ABB RAPID module: Head_Data.mod

MODULE Head_Data
    RECORD breakpoint
        pos Position;
        num Angle;
    ENDRECORD

    RECORD corrorder
        num X_Init;
        num X_StartOffset;
        num X_Depth;
        num X_ReturnLength;
        num Y_StartOffset;
        num Y_Depth;
        num Y_ReturnLength;
        num Z_StartOffset;
        num Z_Depth;
        num Z_ReturnLength;
        num RY_Torch;
        num Y_MoveCorrConnect;
        num Z_MoveCorrConnect;
    ENDRECORD

    RECORD monRobs
        extjoint monExt;
        robjoint monJoint1;
        robjoint monJoint2;
        pose monPose1;
        pose monPose2;
    ENDRECORD

    RECORD edgedata
        pos EdgePos;
        num Height;
        num Breadth;
        num HoleSize;
        num Thickness;
        num AngleHeight;
        num AngleWidth;
    ENDRECORD

    RECORD jointgroup
        jointtarget Joint1;
        jointtarget Joint2;
        jointtarget JointG;
    ENDRECORD

    RECORD pointgroup
        robtarget Point1;
        robtarget Point2;
        robtarget PointG;
    ENDRECORD

    RECORD targetdata
        robtarget position;
        num cpm;
        num schedule;
        num voltage;
        num wfs;
        num Current;
        num WeaveShape;
        num WeaveType;
        num WeaveLength;
        num WeaveWidth;
        num WeaveDwellLeft;
        num WeaveDwellRight;
        num TrackType;
        num TrackGainY;
        num TrackGainZ;
        num MaxCorr;
        num Bias;
    ENDRECORD

    RECORD torchmotion
        num No;
        num LengthOffset;
        num BreadthOffset;
        num HeightOffset;
        num WorkingAngle;
        num TravelAngle;
        num WeldingSpeed;
        num Schedule;
        num Voltage;
        num FeedingSpeed;
        num Current;
        num WeaveShape;
        num WeaveType;
        num WeaveLength;
        num WeaveWidth;
        num WeaveDwellLeft;
        num WeaveDwellRight;
        num TrackType;
        num TrackGainY;
        num TrackGainZ;
        num MaxCorr;
        num Bias;
    ENDRECORD

    RECORD TcpOrder
        num Tcp_X;
        num Tcp_Y;
        num Tcp_Z;
        num Tcp_Angle;
    ENDRECORD

    PERS corrorder corrStart{10}:=[[25,15,30,10,15,40,10,15,30,15,2,20,20],[50,15,30,10,15,40,10,15,30,15,0,20,20],[25,-15,-30,-10,15,40,10,15,30,15,2,20,20],[0,0,0,0,15,40,10,15,30,15,0,20,20],[0,0,0,0,15,40,10,15,40,15,5,20,20],[25,-15,-30,-10,15,40,10,15,30,15,0,20,20],[999,0,0,0,0,0,0,0,0,0,0,0,0],[999,0,0,0,0,0,0,0,0,0,0,0,0],[999,0,0,0,25,40,10,15,30,30,10,0,0],[999,0,0,0,0,0,0,0,0,0,0,0,0]];
    PERS corrorder corrEnd{10}:=[[25,15,30,10,15,40,10,15,30,15,2,20,20],[50,15,30,10,15,40,10,15,30,15,0,20,20],[25,-15,-30,-10,15,40,10,15,30,15,2,20,20],[0,0,0,0,15,40,10,15,30,15,0,20,20],[0,0,0,0,15,40,10,15,40,15,3,20,20],[25,-15,-30,-10,15,40,10,15,30,15,0,20,20],[999,0,0,0,25,40,10,15,30,10,0,0,0],[999,0,0,0,0,0,0,0,0,0,0,0,0],[0,0,0,0,15,40,10,15,30,15,0,20,20],[0,0,0,0,0,0,0,0,0,0,0,20,20]];

    PERS tooldata tWeld:=[TRUE,[[320.377,0,330.247],[0.92587,0,0.37784,0]],[3.1,[-71.4,3.8,173.2],[1,0,0,0],0.055,0.049,0.005]];
    PERS tooldata tWeld1:=[TRUE,[[319.938,-6.311,330],[0.92587,0.003729,0.377818,-0.009129]],[3.1,[-71.4,3.8,173.2],[1,0,0,0],0.055,0.049,0.005]];
    PERS tooldata tWeld2:=[TRUE,[[319.938,-6.311,330],[0.92587,0.003729,0.377818,-0.009128]],[3.1,[-71.4,3.8,173.2],[1,0,0,0],0.055,0.049,0.005]];

    PERS wobjdata WobjFloor:=[FALSE,TRUE,"",[[-9600,5300,2095],[0,1,0,0]],[[0,0,0],[1,0,0,0]]];
    PERS wobjdata wobjWeldLine:=[FALSE,TRUE,"",[[-9600,5300,2095],[0,1,0,0]],[[19996.2,2781.64,4.14455],[0.708156,0.000193577,0.000194152,-0.706056]]];
    ! [PlanB Moving WObj] ELM_X(갠트리 선형축) 연동 좌표계 — 2026-03-05
    ! 변경 전: ufprog=TRUE(고정), ufmec=""  → 갠트리 이동 시 WObj 미추종
    ! 변경 후: ufprog=FALSE(이동), ufmec="ELM_X" → 갠트리와 함께 WObj 이동
    ! uframe: ELM_X 원점 기준(동일), oframe: 기존 uframe 오프셋을 oframe으로 이전
    PERS wobjdata wobjWeldLine1:=[FALSE,FALSE,"ELM_X",[[0,0,0],[1,0,0,0]],[[488,50,1620],[0,0.707107,-0.707107,0]]];
    PERS wobjdata wobjWeldLine2:=[FALSE,FALSE,"ELM_X",[[0,0,0],[1,0,0,0]],[[488,-50,1620],[0,0.707107,0.707107,0]]];
    PERS wobjdata wobjRotCtr1:=[FALSE,TRUE,"",[[488,0,0],[0,0.707107,-0.707107,0]],[[0,0,0],[1,0,0,0]]];
    PERS wobjdata wobjRotCtr2:=[FALSE,TRUE,"",[[488,0,0],[0,0.707107,0.707107,0]],[[0,0,0],[1,0,0,0]]];

    !!! Mechanical Geometry !!!
    PERS num nLimitX_Negative:=-9600;
    PERS num nLimitX_Positive:=12400;
    PERS num nLimitY_Negative:=0;
    PERS num nLimitY_Positive:=5300;
    PERS num nLimitZ_Negative:=0;
    PERS num nLimitZ_Positive:=2095;
    PERS num nLimitR_Negative:=-90;
    PERS num nLimitR_Positive:=90;

    ! HomeGantry Home Information
    PERS num nHomeGantryX:=-9600;
    PERS num nHomeGantryY:=5300;
    PERS num nHomeGantryZ:=2095;
    PERS num nHomeGantryR:=0;

    PERS num nHomeTcpX:=-9600;
    PERS num nHomeTcpY:=5300;
    PERS num nHomeTcpZ:=2095;

    ! LDS Check Calibration Reference Point
    PERS num nHomeAdjustX:=0;
    PERS num nHomeAdjustY:=0;
    PERS num nHomeAdjustZ:=0;
    PERS num nHomeAdjustR:=0;

    PERS num Camera_Door:=0;
    PERS num Camera_Tilt:=0;

    ! Robot Welding Posture Height
    PERS num nRobHeightMin:=1100;
    PERS num nRobCorrSpaceHeight:=1680;
    PERS num nRobWorkSpaceHeight:=1680;
    PERS num nRobWeldSpaceHeight:=1620;

    PERS num nRotationNegLimit:=-90;
    PERS num nRotationPosLimit:=90;

    !! Variables for Commands
    PERS num nCmdInput:=0;
    PERS num nCmdOutput:=0;
    PERS num nCmdMatch:=0;


    !!! Bool Data !!!
    PERS bool bEnableWeldSkip:=FALSE;
    PERS bool bEnableStartEndPointCorr:=FALSE;
    PERS bool bEnableManualMacro:=FALSE;
    PERS bool bWireTouch1;
    PERS bool bWireTouch2;
    PERS bool bRobSwap:=FALSE;

    !!!!  WarmUp_X !!!!!
    CONST num nWarmUp_Target_X:=10000;

    !commands for move
    CONST num CMD_MOVE_TO_WORLDHOME:=101;
    CONST num CMD_MOVE_TO_MeasurementHOME:=102;
    CONST num CMD_MOVE_TO_TEACHING_All:=104;
    CONST num CMD_MOVE_TO_TEACHING_R1:=105;
    CONST num CMD_MOVE_TO_TEACHING_R2:=106;
    CONST num CMD_MOVE_JOINTS:=107;
    CONST num CMD_MOVE_ABS_GANTRY:=108;
    CONST num CMD_MOVE_INC_GANTRY:=109;
    CONST num CMD_MOVE_TO_ZHOME:=110;
    CONST num CMD_MOVE_TO_nWarmUp:=112;
    CONST num CMD_Tcp_Inspect:=151;

    ! commands for welding
    CONST num CMD_WELD:=200;
    CONST num CMD_WELD_MOTION:=201;
    CONST num CMD_WELD_CORR:=202;
    CONST num CMD_WELD_MOTION_CORR:=203;
    CONST num CMD_WELD_MM:=204;
    CONST num CMD_WELD_MOTION_MM:=205;
    CONST num CMD_WELD_CORR_MM:=206;
    CONST num CMD_WELD_MOTION_CORR_MM:=207;

    !commands for camera actions
    CONST num CMD_CAMERA_DOOR_OPEN:=301;
    CONST num CMD_CAMERA_DOOR_CLOSE:=302;
    CONST num CMD_CAMERA_BLOW_ON:=303;
    CONST num CMD_CAMERA_BLOW_OFF:=304;
    CONST num CMD_CAMERA1_DOOR_OPEN:=311;
    CONST num CMD_CAMERA1_DOOR_CLOSE:=312;
    CONST num CMD_CAMERA2_DOOR_OPEN:=321;
    CONST num CMD_CAMERA2_DOOR_CLOSE:=322;
    CONST num CMD_CAMERA1_BLOW_ON:=313;
    CONST num CMD_CAMERA2_BLOW_ON:=323;
    CONST num CMD_CAMERA1_BLOW_OFF:=314;
    CONST num CMD_CAMERA2_BLOW_OFF:=324;

    !commands for wire processing
    CONST num CMD_WIRE_CUT:=501;
    CONST num CMD_WIRE_CLEAN:=502;
    CONST num CMD_WIRE_BULLSEYE_CHECK:=505;
    CONST num CMD_WIRE_BULLSEYE_UPDATE:=506;
    CONST num CMD_WIRE_ReplacementMode:=507;
    CONST num CMD_ROB1_WIRE_CUT:=511;
    CONST num CMD_ROB2_WIRE_CUT:=512;
    CONST num CMD_WIRE_CLEAN_R1:=513;
    CONST num CMD_WIRE_CLEAN_R2:=514;

    CONST num CMD_GotoTeachingToWirecut:=551;
    CONST num CMD_TeachingToWirecutEntry_R1:=552;
    CONST num CMD_TeachingToWirecut_R1:=553;
    CONST num CMD_ReturnToWirecut:=554;
    CONST num CMD_TeachingToWirecutEntry_R2:=562;
    CONST num CMD_TeachingToWirecut_R2:=563;

    !commands for gantry mechanical origin checking
    CONST num CMD_HOLE_CHECK:=601;
    CONST num CMD_LDS_CHECK:=602;
    CONST num CMD_ManualOrigin_CHECK:=603;

    ! variables related to commands
    PERS num Command:=0;

    !Weld Time
    VAR clock clockWeldTime;
    PERS num nclockWeldTime{2}:=[270.196,134.768];

    !Cycle Time
    VAR clock clockCycleTime;
    PERS num nclockCycleTime:=334.572;

    PERS num nCameraRotationAngle:=0;

    ! variables for welding command
    PERS num nMotionStep:=5;
    PERS num nMotionTotalStep{2}:=[8,8];
    PERS num nMotionStepCount{2}:=[10,10];

    PERS num nLengthWeldLine:=2662.05;
    PERS num nOffsetLength:=0;
    PERS num nOffsetLengthBuffer:=10;

    !! Variables for Welding Macro
    !! sMacro 2nd,3rd Dim: (1: Open, 2: Snip, 3: Welding, 4: Continued, 5: Divied, 8:MergeStart, 9:MergeEnd)
    PERS string stMacro{2}:=["244","244"];
    PERS string stMacroBuffer_{2};
    PERS num nMacro100{2}:=[2,2];
    PERS num nMacro010{2}:=[4,4];
    PERS num nMacro001{2}:=[4,4];
    PERS num nMacro{2}:=[244,244];

    PERS num nMotionStartStepLast{2}:=[4,4];
    PERS num nMotionEndStepLast{2}:=[4,4];
    PERS num nRunningStep{2}:=[40,40];

    PERS edgedata edgeStart{2}:=[[[20002.2,2781.66,4.15085],50,50,0,12,0,0],[[19990.2,2781.62,4.13825],50,50,0,12,0,0]];
    PERS edgedata edgeEnd{2}:=[[[20010.1,119.623,2.69116],50,50,0,12,0,0],[[19998.1,119.588,2.67856],50,50,0,12,0,0]];

    PERS pos posNull:=[0,0,0];
    PERS pos posStart:=[19996.4,2781.64,5.3429];
    PERS pos posStartLast:=[19996.4,2781.64,5.3429];
    PERS num nStartThick:=14.0106;
    PERS pos posEnd:=[20000.3,119.594,0.735352];
    PERS pos posEndLast:=[20000.3,119.594,0.735352];
    PERS num nEndThick:=13.2815;

    PERS breakpoint BreakPoints{10}:=[[[0,0,0],0],[[0,0,0],0],[[0,0,0],0],[[0,0,0],0],[[0,0,0],0],[[0,0,0],0],[[0,0,0],0],[[0,0,0],0],[[0,0,0],0],[[0,0,0],0]];

    ! data for z pos optimization [move,enter,exit]
    PERS num nMaxPartHeightNearArray{3}:=[300,300,300];

    PERS num nTempAdjustGantryZ;

    !!! Variable for correction weldline start & end Pos !!!
    CONST bool bStart:=TRUE;
    CONST bool bEnd:=FALSE;
    PERS bool bCorrectionOk:=FALSE;
    PERS bool bPlateTiltedRx:=FALSE;
    PERS robtarget pSearchStart:=[[-15,6.31316,14.5561],[0.208209,0.745508,-0.572049,0.271343],[0,0,0,1],[9E+09,9E+09,9E+09,9E+09,9E+09,9E+09]];
    PERS robtarget pSearchEnd:=[[15,6.31316,14.5561],[0.208209,0.745508,-0.572049,0.271343],[0,0,0,1],[9E+09,9E+09,9E+09,9E+09,9E+09,9E+09]];
    PERS num nCorrZ_Store:=5.43813;
    PERS num nCorrY_Store:=1.20374;
    PERS num nCorrX_Store:=-5.98633;
    PERS num nCorrFailOffs:=0;
    PERS pos pCorredPosBuffer:=[13.5035,6.32969,14.5309];
    PERS pos pCorredStartPos{2}:=[[2086.6,5904.59,39.6865],[2086.6,5904.59,39.6865]];
    PERS pos pCorredEndPos{2}:=[[2082.19,4521.61,35.0346],[2086.6,5904.59,39.6865]];
    PERS pos pCorredSplitPos:=[2082.19,4521.61,35.0346];

    PERS bool bWeldLineLengthCalc:=FALSE;
    PERS bool bMoveGantry:=FALSE;

    !! Variables for Position of Gantry Move
    PERS extjoint extGantryPos:=[13750,2300,2100,0,0,13750];

    !!! RoboTarget !!!
    CONST robtarget pNull:=[[0,0,0],[1,0,0,0],[0,0,0,0],[9E+09,9E+09,9E+09,9E+09,9E+09,9E+09]];
    CONST robtarget pHome:=[[423.10464973,-0.304,-470.07267919],[0.342020143,0,-0.939692621,0],[0,0,-1,0],[0,0,0,9E+09,9E+09,9E+09]];

    PERS robtarget pReadyConf{2}:=[[[200.384,-150.531,462.112],[0.16437,-0.687406,-0.687732,-0.165769],[0,-1,0,1],[-8705.17,-8705.17,300.411,482.178,9E+09,9E+09]],[[200.384,-150.531,462.112],[0.16437,-0.687406,-0.687732,-0.165769],[0,-1,0,1],[-8705.17,-8705.17,300.411,482.178,9E+09,9E+09]]];
    PERS robtarget pTargetWeldArray{30}:=[[[-5,5,5],[0.307623,-0.549545,-0.742667,-0.227629],[0,0,0,0],[1400,1400,1200,0,9E+9,9E+9]],[[-5,-6,5],[0.307623,-0.549545,-0.742667,-0.227629],[0,0,0,0],[1400,1400,1200,0,9E+9,9E+9]],[[4,-3,5],[0.307623,-0.549545,-0.742667,-0.227629],[0,0,0,0],[1400,1400,1200,0,9E+9,9E+9]],[[200,-3,5],[0.270598,-0.653282,-0.653282,-0.270598],[0,0,0,0],[1400,1400,1200,0,9E+9,9E+9]],[[800,-3,5],[0.270598,-0.653282,-0.653282,-0.270598],[0,0,0,0],[1400,1400,1800,0,9E+9,9E+9]],[[951,-3,5],[0.270598,-0.653282,-0.653282,-0.270598],[0,0,0,0],[1400,1400,1800,0,9E+9,9E+9]],[[986,-3,5],[0.270598,-0.653282,-0.653282,-0.270598],[0,0,0,0],[1400,1400,1800,0,9E+9,9E+9]],[[1002,-3,5],[0.227629,-0.742667,-0.549545,-0.307623],[0,0,0,0],[1400,1400,1800,0,9E+9,9E+9]],[[1005,-6,5],[0.227629,-0.742667,-0.549545,-0.307623],[0,0,0,0],[1400,1400,1800,0,9E+9,9E+9]],[[1005,7,5],[0.227629,-0.742667,-0.549545,-0.307623],[0,0,0,0],[1400,1400,1800,0,9E+9,9E+9]],
                                         [[1005,-6,5],[0.227629,-0.742667,-0.549545,-0.307623],[0,0,0,0],[1400,1400,1800,0,9E+9,9E+9]],[[951,-3,5],[0.270598,-0.653282,-0.653282,-0.270598],[0,0,0,0],[1400,1400,1800,0,9E+9,9E+9]],[[0,0,0],[1,0,0,0],[0,0,0,0],[0,0,0,0,9E+9,9E+9]],[[0,0,0],[1,0,0,0],[0,0,0,0],[0,0,0,0,9E+9,9E+9]],[[0,0,0],[1,0,0,0],[0,0,0,0],[0,0,0,0,9E+9,9E+9]],[[0,0,0],[1,0,0,0],[0,0,0,0],[0,0,0,0,9E+9,9E+9]],[[0,0,0],[1,0,0,0],[0,0,0,0],[0,0,0,0,9E+9,9E+9]],[[0,0,0],[1,0,0,0],[0,0,0,0],[0,0,0,0,9E+9,9E+9]],[[0,0,0],[1,0,0,0],[0,0,0,0],[0,0,0,0,9E+9,9E+9]],[[0,0,0],[1,0,0,0],[0,0,0,0],[0,0,0,0,9E+9,9E+9]],
                                         [[0,0,0],[1,0,0,0],[0,0,0,0],[0,0,0,0,9E+9,9E+9]],[[0,0,0],[1,0,0,0],[0,0,0,0],[0,0,0,0,9E+9,9E+9]],[[0,0,0],[1,0,0,0],[0,0,0,0],[0,0,0,0,9E+9,9E+9]],[[0,0,0],[1,0,0,0],[0,0,0,0],[0,0,0,0,9E+9,9E+9]],[[0,0,0],[1,0,0,0],[0,0,0,0],[0,0,0,0,9E+9,9E+9]],[[0,0,0],[1,0,0,0],[0,0,0,0],[0,0,0,0,9E+9,9E+9]],[[0,0,0],[1,0,0,0],[0,0,0,0],[0,0,0,0,9E+9,9E+9]],[[0,0,0],[1,0,0,0],[0,0,0,0],[0,0,0,0,9E+9,9E+9]],[[0,0,0],[1,0,0,0],[0,0,0,0],[0,0,0,0,9E+9,9E+9]],[[0,0,0],[1,0,0,0],[0,0,0,0],[0,0,0,0,9E+9,9E+9]]];

    !!! Joint Target !!!
    PERS jointtarget jNull:=[[0,0,0,0,0,0],[0,0,0,0,9E+09,0]];
    PERS jointtarget jHomeJoint:=[[9E+09,9E+09,9E+09,9E+09,9E+09,9E+09],[8000,5300,0,0,9E+09,8000]];
    PERS jointgroup jgHomeJoint:=[[[90,90,-45,0,20,0],[9E+09,9E+09,9E+09,9E+09,9E+09,9E+09]],[[90,90,-45,0,20,0],[9E+09,9E+09,9E+09,9E+09,9E+09,9E+09]],[[9E+09,9E+09,9E+09,9E+09,9E+09,9E+09],[8000,5300,0,0,9E+09,8000]]];
    PERS jointtarget jHomeJointBackup:=[[9E+09,9E+09,9E+09,9E+09,9E+09,9E+09],[0,0,6000,500,9E+09,9E+09]];
    PERS jointtarget jRepairJoint:=[[9E+09,9E+09,9E+09,9E+09,9E+09,9E+09],[0,0,6000,500,9E+09,9E+09]];
    PERS jointtarget jMoveReady:=[[9E+9,9E+9,9E+9,9E+9,9E+9,9E+9],[-8707.81,-8707.8,1477.15,0,9E+9,9E+9]];

    PERS jointtarget jJointStepArray{10}:=[[[0,0,0,0,0,0],[0,0,0,0,0,0]],[[0,0,0,0,0,0],[0,0,0,0,0,0]],[[0,0,0,0,0,0],[0,0,0,0,0,0]],[[0,0,0,0,0,0],[0,0,0,0,0,0]],[[0,0,0,0,0,0],[0,0,0,0,0,0]],[[0,-95,65,0,-35,0],[0,0,0,0,0,0]],[[0,0,0,0,0,0],[0,0,0,0,0,0]],[[0,0,0,0,0,0],[0,0,0,0,0,0]],[[0,0,0,0,0,0],[0,0,0,0,0,0]],[[0,-46.86,14,0,-57.52,1.03],[0,0,0,0,0,0]]];

    PERS jointtarget jWeldPos{40}:=[[[0,0,0,0,0,0],[0,0,0,0,9E+09,9E+09]],[[0,0,0,0,0,0],[0,0,0,0,9E+09,9E+09]],[[0,0,0,0,0,0],[0,0,0,0,9E+09,9E+09]],[[0,0,0,0,0,0],[0,0,0,0,9E+09,9E+09]],[[0,0,0,0,0,0],[0,0,0,0,9E+09,9E+09]],[[0,0,0,0,0,0],[0,0,0,0,9E+09,9E+09]],[[0,0,0,0,0,0],[0,0,0,0,9E+09,9E+09]],[[0,0,0,0,0,0],[0,0,0,0,9E+09,9E+09]],[[0,0,0,0,0,0],[0,0,0,0,9E+09,9E+09]],[[0,0,0,0,0,0],[0,0,0,0,9E+09,9E+09]],[[0,0,0,0,0,0],[0,0,0,0,9E+09,9E+09]],[[0,0,0,0,0,0],[0,0,0,0,9E+09,9E+09]],[[0,0,0,0,0,0],[0,0,0,0,9E+09,9E+09]],[[0,0,0,0,0,0],[0,0,0,0,9E+09,9E+09]],[[0,0,0,0,0,0],[0,0,0,0,9E+09,9E+09]],[[0,0,0,0,0,0],[0,0,0,0,9E+09,9E+09]],[[0,0,0,0,0,0],[0,0,0,0,9E+09,9E+09]],[[0,0,0,0,0,0],[0,0,0,0,9E+09,9E+09]],[[0,0,0,0,0,0],[0,0,0,0,9E+09,9E+09]],[[0,0,0,0,0,0],[0,0,0,0,9E+09,9E+09]],[[0,0,0,0,0,0],[0,0,0,0,9E+09,9E+09]],[[0,0,0,0,0,0],[0,0,0,0,9E+09,9E+09]],[[0,0,0,0,0,0],[0,0,0,0,9E+09,9E+09]],[[0,0,0,0,0,0],[0,0,0,0,9E+09,9E+09]],[[0,0,0,0,0,0],[0,0,0,0,9E+09,9E+09]],[[0,0,0,0,0,0],[0,0,0,0,9E+09,9E+09]],[[0,0,0,0,0,0],[0,0,0,0,9E+09,9E+09]],[[0,0,0,0,0,0],[0,0,0,0,9E+09,9E+09]],[[0,0,0,0,0,0],[0,0,0,0,9E+09,9E+09]],[[0,0,0,0,0,0],[0,0,0,0,9E+09,9E+09]],[[0,0,0,0,0,0],[0,0,0,0,9E+09,9E+09]],[[0,0,0,0,0,0],[0,0,0,0,9E+09,9E+09]],[[0,0,0,0,0,0],[0,0,0,0,9E+09,9E+09]],[[0,0,0,0,0,0],[0,0,0,0,9E+09,9E+09]],[[0,0,0,0,0,0],[0,0,0,0,9E+09,9E+09]],[[0,0,0,0,0,0],[0,0,0,0,9E+09,9E+09]],[[0,0,0,0,0,0],[0,0,0,0,9E+09,9E+09]],[[0,0,0,0,0,0],[0,0,0,0,9E+09,9E+09]],[[0,0,0,0,0,0],[0,0,0,0,9E+09,9E+09]],[[0,0,0,0,0,0],[0,0,0,0,9E+09,9E+09]]];
    PERS jointtarget jTest1:=[[9E+09,9E+09,9E+09,9E+09,9E+09,9E+09],[0,0,0,0,9E+09,0]];
    PERS jointtarget jTest2:=[[9E+09,9E+09,9E+09,9E+09,9E+09,9E+09],[0,0,0,0,9E+09,0]];
    PERS jointtarget jTest3:=[[9E+09,9E+09,9E+09,9E+09,9E+09,9E+09],[0,0,0,0,9E+09,0]];
    PERS jointtarget jTest4:=[[9E+09,9E+09,9E+09,9E+09,9E+09,9E+09],[0,0,0,0,9E+09,0]];

    !!! Variables for macroReference !!!
    PERS torchmotion macroAutoStartA{2,10}:=[[[1,0,-2,2,50,0,60,5,36.8,230,380,1,2,2,1.5,1,1,0,0,0,0,0],[2,1,-2,2,50,0,60,5,36.8,230,380,1,2,2,1.5,1,1,0,0,0,0,0],[3,2,-2,2,50,0,60,5,36.8,230,380,1,2,2,1.5,1,1,0,0,0,0,0],[4,3,-2,2,50,0,60,5,36.8,230,380,1,2,2,1.5,1,1,0,0,0,0,0],[999,1,1,1,1,1,1,1,1,1,1,1,1,1,1,1,1,1,1,1,1,1],[1,1,1,1,1,1,1,1,1,1,1,1,1,1,1,1,1,1,1,1,1,1],[1,1,1,1,1,1,1,1,1,1,1,1,1,1,1,1,1,1,1,1,1,1],[1,1,1,1,1,1,1,1,1,1,1,1,1,1,1,1,1,1,1,1,1,1],[1,1,1,1,1,1,1,1,1,1,1,1,1,1,1,1,1,1,1,1,1,1],[1,1,1,1,1,1,1,1,1,1,1,1,1,1,1,1,1,1,1,1,1,1]],[[1,0,-3,2,50,0,60,5,36.3,232,360,1,2,2,1.5,1,1,0,0,0,0,0],[2,1,-3,2,50,0,60,5,36.3,232,360,1,2,2,1.5,1,1,0,0,0,0,0],[3,2,-3,2,50,0,60,5,36.3,232,360,1,2,2,1.5,1,1,0,0,0,0,0],[4,3,-3,2,50,0,60,5,36.3,232,360,1,2,2,1.5,1,1,0,0,0,0,0],[999,1,1,1,1,1,1,1,1,1,1,1,1,1,1,1,1,1,1,1,1,1],[1,1,1,1,1,1,1,1,1,1,1,1,1,1,1,1,1,1,1,1,1,1],[1,1,1,1,1,1,1,1,1,1,1,1,1,1,1,1,1,1,1,1,1,1],[1,1,1,1,1,1,1,1,1,1,1,1,1,1,1,1,1,1,1,1,1,1],[1,1,1,1,1,1,1,1,1,1,1,1,1,1,1,1,1,1,1,1,1,1],[1,1,1,1,1,1,1,1,1,1,1,1,1,1,1,1,1,1,1,1,1,1]]];
    PERS torchmotion macroAutoStartB{2,10}:=[[[1,0,-2,2,50,0,60,5,36.8,230,380,1,2,2,1.5,1,1,0,0,0,0,0],[2,1,-2,2,50,0,60,5,36.8,230,380,1,2,2,1.5,1,1,0,0,0,0,0],[3,2,-2,2,50,0,60,5,36.8,230,380,1,2,2,1.5,1,1,0,0,0,0,0],[4,3,-2,2,50,0,60,5,36.8,230,380,1,2,2,1.5,1,1,0,0,0,0,0],[999,1,1,1,1,1,1,1,1,1,1,1,1,1,1,1,1,1,1,1,1,1],[1,1,1,1,1,1,1,1,1,1,1,1,1,1,1,1,1,1,1,1,1,1],[1,1,1,1,1,1,1,1,1,1,1,1,1,1,1,1,1,1,1,1,1,1],[1,1,1,1,1,1,1,1,1,1,1,1,1,1,1,1,1,1,1,1,1,1],[1,1,1,1,1,1,1,1,1,1,1,1,1,1,1,1,1,1,1,1,1,1],[1,1,1,1,1,1,1,1,1,1,1,1,1,1,1,1,1,1,1,1,1,1]],[[1,0,-3,2,50,0,60,5,36.3,232,360,1,2,2,1.5,1,1,0,0,0,0,0],[2,1,-3,2,50,0,60,5,36.3,232,360,1,2,2,1.5,1,1,0,0,0,0,0],[3,2,-3,2,50,0,60,5,36.3,232,360,1,2,2,1.5,1,1,0,0,0,0,0],[4,3,-3,2,50,0,60,5,36.3,232,360,1,2,2,1.5,1,1,0,0,0,0,0],[999,1,1,1,1,1,1,1,1,1,1,1,1,1,1,1,1,1,1,1,1,1],[1,1,1,1,1,1,1,1,1,1,1,1,1,1,1,1,1,1,1,1,1,1],[1,1,1,1,1,1,1,1,1,1,1,1,1,1,1,1,1,1,1,1,1,1],[1,1,1,1,1,1,1,1,1,1,1,1,1,1,1,1,1,1,1,1,1,1],[1,1,1,1,1,1,1,1,1,1,1,1,1,1,1,1,1,1,1,1,1,1],[1,1,1,1,1,1,1,1,1,1,1,1,1,1,1,1,1,1,1,1,1,1]]];
    PERS torchmotion macroAutoEndA{2,10}:=[[[1,-3,-2,2,50,0,60,5,36.8,230,380,1,2,2,1.5,1,1,0,10,20,30,0],[2,-2,-2,2,50,0,60,5,36.8,230,380,1,2,2,1.5,1,1,0,0,0,0,0],[3,-1,-2,2,50,0,60,5,36.8,230,380,1,2,2,1.5,1,1,0,0,0,0,0],[4,0,-2,2,50,0,60,5,36.8,230,380,1,2,2,1.5,1,1,0,0,0,0,0],[999,1,1,1,1,1,1,1,1,1,1,1,1,1,1,1,1,1,1,1,1,1],[1,1,1,1,1,1,1,1,1,1,1,1,1,1,1,1,1,1,1,1,1,1],[1,1,1,1,1,1,1,1,1,1,1,1,1,1,1,1,1,1,1,1,1,1],[1,1,1,1,1,1,1,1,1,1,1,1,1,1,1,1,1,1,1,1,1,1],[1,1,1,1,1,1,1,1,1,1,1,1,1,1,1,1,1,1,1,1,1,1],[1,1,1,1,1,1,1,1,1,1,1,1,1,1,1,1,1,1,1,1,1,1]],[[1,-3,-3,2,50,0,60,5,36.3,232,360,1,2,2,1.5,1,1,0,10,20,30,0],[2,-2,-3,2,50,0,60,5,36.3,232,360,1,2,2,1.5,1,1,0,0,0,0,0],[3,-1,-2,2,50,0,60,5,36.3,232,360,1,2,2,1.5,1,1,0,0,0,0,0],[4,0,-2,2,50,0,60,5,36.3,232,360,1,2,2,1.5,1,1,0,0,0,0,0],[999,1,1,1,1,1,1,1,1,1,1,1,1,1,1,1,1,1,1,1,1,1],[1,1,1,1,1,1,1,1,1,1,1,1,1,1,1,1,1,1,1,1,1,1],[1,1,1,1,1,1,1,1,1,1,1,1,1,1,1,1,1,1,1,1,1,1],[1,1,1,1,1,1,1,1,1,1,1,1,1,1,1,1,1,1,1,1,1,1],[1,1,1,1,1,1,1,1,1,1,1,1,1,1,1,1,1,1,1,1,1,1],[1,1,1,1,1,1,1,1,1,1,1,1,1,1,1,1,1,1,1,1,1,1]]];
    PERS torchmotion macroAutoEndB{2,10}:=[[[1,-3,-2,2,50,0,60,5,36.8,230,380,1,2,2,1.5,1,1,0,10,20,30,0],[2,-2,-2,2,50,0,60,5,36.8,230,380,1,2,2,1.5,1,1,0,0,0,0,0],[3,-1,-2,2,50,0,60,5,36.8,230,380,1,2,2,1.5,1,1,0,0,0,0,0],[4,0,-2,2,50,0,60,5,36.8,230,380,1,2,2,1.5,1,1,0,0,0,0,0],[999,1,1,1,1,1,1,1,1,1,1,1,1,1,1,1,1,1,1,1,1,1],[1,1,1,1,1,1,1,1,1,1,1,1,1,1,1,1,1,1,1,1,1,1],[1,1,1,1,1,1,1,1,1,1,1,1,1,1,1,1,1,1,1,1,1,1],[1,1,1,1,1,1,1,1,1,1,1,1,1,1,1,1,1,1,1,1,1,1],[1,1,1,1,1,1,1,1,1,1,1,1,1,1,1,1,1,1,1,1,1,1],[1,1,1,1,1,1,1,1,1,1,1,1,1,1,1,1,1,1,1,1,1,1]],[[1,-3,-3,2,50,0,60,5,36.3,232,360,1,2,2,1.5,1,1,0,10,20,30,0],[2,-2,-3,2,50,0,60,5,36.3,232,360,1,2,2,1.5,1,1,0,0,0,0,0],[3,-1,-2,2,50,0,60,5,36.3,232,360,1,2,2,1.5,1,1,0,0,0,0,0],[4,0,-2,2,50,0,60,5,36.3,232,360,1,2,2,1.5,1,1,0,0,0,0,0],[999,1,1,1,1,1,1,1,1,1,1,1,1,1,1,1,1,1,1,1,1,1],[1,1,1,1,1,1,1,1,1,1,1,1,1,1,1,1,1,1,1,1,1,1],[1,1,1,1,1,1,1,1,1,1,1,1,1,1,1,1,1,1,1,1,1,1],[1,1,1,1,1,1,1,1,1,1,1,1,1,1,1,1,1,1,1,1,1,1],[1,1,1,1,1,1,1,1,1,1,1,1,1,1,1,1,1,1,1,1,1,1],[1,1,1,1,1,1,1,1,1,1,1,1,1,1,1,1,1,1,1,1,1,1]]];

    PERS torchmotion macroManualStartA{2,10}:=[[[1,0,-2,2,50,0,60,5,36.5,230,380,1,2,2,1.5,1,1,0,0,0,0,0],[2,1,-2,2,50,0,60,5,36.5,230,380,1,2,2,1.5,1,1,0,0,0,0,0],[3,2,-2,2,50,0,60,5,36.5,230,380,1,2,2,1.5,1,1,0,0,0,0,0],[4,3,-2,2,50,0,60,5,36.5,230,380,1,2,2,1.5,1,1,0,0,0,0,0],[999,1,1,1,1,1,1,1,1,1,1,1,1,1,1,1,1,1,1,1,1,1],[1,1,1,1,1,1,1,1,1,1,1,1,1,1,1,1,1,1,1,1,1,1],[1,1,1,1,1,1,1,1,1,1,1,1,1,1,1,1,1,1,1,1,1,1],[1,1,1,1,1,1,1,1,1,1,1,1,1,1,1,1,1,1,1,1,1,1],[1,1,1,1,1,1,1,1,1,1,1,1,1,1,1,1,1,1,1,1,1,1],[1,1,1,1,1,1,1,1,1,1,1,1,1,1,1,1,1,1,1,1,1,1]],[[1,0,-3,2,50,0,60,5,36.3,232,360,1,2,2,1.5,1,1,0,0,0,0,0],[2,1,-3,2,50,0,60,5,36.3,232,360,1,2,2,1.5,1,1,0,0,0,0,0],[3,2,-3,2,50,0,60,5,36.3,232,360,1,2,2,1.5,1,1,0,0,0,0,0],[4,3,-3,2,50,0,60,5,36.3,232,360,1,2,2,1.5,1,1,0,0,0,0,0],[999,1,1,1,1,1,1,1,1,1,1,1,1,1,1,1,1,1,1,1,1,1],[1,1,1,1,1,1,1,1,1,1,1,1,1,1,1,1,1,1,1,1,1,1],[1,1,1,1,1,1,1,1,1,1,1,1,1,1,1,1,1,1,1,1,1,1],[1,1,1,1,1,1,1,1,1,1,1,1,1,1,1,1,1,1,1,1,1,1],[1,1,1,1,1,1,1,1,1,1,1,1,1,1,1,1,1,1,1,1,1,1],[1,1,1,1,1,1,1,1,1,1,1,1,1,1,1,1,1,1,1,1,1,1]]];
    ![[[1,0,-2,2,50,38,60,5,36.5,230,370,1,2,2,2,1,1,0,0,0,0,0],[2,0,-2,2,50,38,60,5,36.5,230,370,1,2,2,2,1,1,0,0,0,0,0],[3,0,-2,2,50,38,60,5,36.5,230,370,1,2,2,2,1,1,0,0,0,0,0],[4,0,-2,2,50,38,60,5,36.5,230,370,1,2,2,2,1,1,0,0,0,0,0],[999,1,1,1,1,1,1,1,1,1,1,1,1,1,1,1,1,1,1,1,1,1],[1,1,1,1,1,1,1,1,1,1,1,1,1,1,1,1,1,1,1,1,1,1],[1,1,1,1,1,1,1,1,1,1,1,1,1,1,1,1,1,1,1,1,1,1],[1,1,1,1,1,1,1,1,1,1,1,1,1,1,1,1,1,1,1,1,1,1],[1,1,1,1,1,1,1,1,1,1,1,1,1,1,1,1,1,1,1,1,1,1],[1,1,1,1,1,1,1,1,1,1,1,1,1,1,1,1,1,1,1,1,1,1]],[[1,0,-2,2,50,38,60,5,36.5,230,360,1,2,2,2,1,1,0,0,0,0,0],[2,0,-2,2,50,38,60,5,36.5,230,360,1,2,2,2,1,1,0,0,0,0,0],[3,0,-2,2,50,38,60,5,36.5,230,360,1,2,2,2,1,1,0,0,0,0,0],[4,0,-2,2,50,38,60,5,36.5,230,360,1,2,2,2,1,1,0,0,0,0,0],[999,1,1,1,1,1,1,1,1,1,1,1,1,1,1,1,1,1,1,1,1,1],[1,1,1,1,1,1,1,1,1,1,1,1,1,1,1,1,1,1,1,1,1,1],[1,1,1,1,1,1,1,1,1,1,1,1,1,1,1,1,1,1,1,1,1,1],[1,1,1,1,1,1,1,1,1,1,1,1,1,1,1,1,1,1,1,1,1,1],[1,1,1,1,1,1,1,1,1,1,1,1,1,1,1,1,1,1,1,1,1,1],[1,1,1,1,1,1,1,1,1,1,1,1,1,1,1,1,1,1,1,1,1,1]]];
    ![[[1,0,-2,2,50,0,60,5,37,230,380,1,2,2,2,1,1,0,0,0,0,0],[2,0,-2,2,50,0,60,5,37,230,380,1,2,2,2,1,1,0,0,0,0,0],[3,0,-2,2,50,0,60,5,37,230,380,1,2,2,2,1,1,0,0,0,0,0],[4,0,-2,2,50,0,60,5,37,230,380,1,2,2,2,1,1,0,0,0,0,0],[999,1,1,1,1,1,1,1,1,1,1,1,1,1,1,1,1,1,1,1,1,1],[1,1,1,1,1,1,1,1,1,1,1,1,1,1,1,1,1,1,1,1,1,1],[1,1,1,1,1,1,1,1,1,1,1,1,1,1,1,1,1,1,1,1,1,1],[1,1,1,1,1,1,1,1,1,1,1,1,1,1,1,1,1,1,1,1,1,1],[1,1,1,1,1,1,1,1,1,1,1,1,1,1,1,1,1,1,1,1,1,1],[1,1,1,1,1,1,1,1,1,1,1,1,1,1,1,1,1,1,1,1,1,1]],[[1,0,-2,2,50,0,60,5,36.5,230,360,1,2,2,2,1,1,0,0,0,0,0],[2,0,-2,2,50,0,60,5,36.5,230,360,1,2,2,2,1,1,0,0,0,0,0],[3,0,-2,2,50,0,60,5,36.5,230,360,1,2,2,2,1,1,0,0,0,0,0],[4,0,-2,2,50,0,60,5,36.5,230,360,1,2,2,2,1,1,0,0,0,0,0],[999,1,1,1,1,1,1,1,1,1,1,1,1,1,1,1,1,1,1,1,1,1],[1,1,1,1,1,1,1,1,1,1,1,1,1,1,1,1,1,1,1,1,1,1],[1,1,1,1,1,1,1,1,1,1,1,1,1,1,1,1,1,1,1,1,1,1],[1,1,1,1,1,1,1,1,1,1,1,1,1,1,1,1,1,1,1,1,1,1],[1,1,1,1,1,1,1,1,1,1,1,1,1,1,1,1,1,1,1,1,1,1],[1,1,1,1,1,1,1,1,1,1,1,1,1,1,1,1,1,1,1,1,1,1]]];
    PERS torchmotion macroManualStartB{2,10}:=[[[1,0,-2,2,50,0,60,5,36.5,230,380,1,2,2,1.5,1,1,0,0,0,0,0],[2,1,-2,2,50,0,60,5,36.5,230,380,1,2,2,1.5,1,1,0,0,0,0,0],[3,2,-2,2,50,0,60,5,36.5,230,380,1,2,2,1.5,1,1,0,0,0,0,0],[4,3,-2,2,50,0,60,5,36.5,230,380,1,2,2,1.5,1,1,0,0,0,0,0],[999,1,1,1,1,1,1,1,1,1,1,1,1,1,1,1,1,1,1,1,1,1],[1,1,1,1,1,1,1,1,1,1,1,1,1,1,1,1,1,1,1,1,1,1],[1,1,1,1,1,1,1,1,1,1,1,1,1,1,1,1,1,1,1,1,1,1],[1,1,1,1,1,1,1,1,1,1,1,1,1,1,1,1,1,1,1,1,1,1],[1,1,1,1,1,1,1,1,1,1,1,1,1,1,1,1,1,1,1,1,1,1],[1,1,1,1,1,1,1,1,1,1,1,1,1,1,1,1,1,1,1,1,1,1]],[[1,0,-3,2,50,0,60,5,36.3,232,360,1,2,2,1.5,1,1,0,0,0,0,0],[2,1,-3,2,50,0,60,5,36.3,232,360,1,2,2,1.5,1,1,0,0,0,0,0],[3,2,-3,2,50,0,60,5,36.3,232,360,1,2,2,1.5,1,1,0,0,0,0,0],[4,3,-3,2,50,0,60,5,36.3,232,360,1,2,2,1.5,1,1,0,0,0,0,0],[999,1,1,1,1,1,1,1,1,1,1,1,1,1,1,1,1,1,1,1,1,1],[1,1,1,1,1,1,1,1,1,1,1,1,1,1,1,1,1,1,1,1,1,1],[1,1,1,1,1,1,1,1,1,1,1,1,1,1,1,1,1,1,1,1,1,1],[1,1,1,1,1,1,1,1,1,1,1,1,1,1,1,1,1,1,1,1,1,1],[1,1,1,1,1,1,1,1,1,1,1,1,1,1,1,1,1,1,1,1,1,1],[1,1,1,1,1,1,1,1,1,1,1,1,1,1,1,1,1,1,1,1,1,1]]];
    ![[[1,0,-2,2,50,0,60,5,37,230,380,1,2,2,2,1,1,0,0,0,0,0],[2,0,-2,2,50,0,60,5,37,230,380,1,2,2,2,1,1,0,0,0,0,0],[3,0,-2,2,50,0,60,5,37,230,380,1,2,2,2,1,1,0,0,0,0,0],[4,0,-2,2,50,0,60,5,37,230,380,1,2,2,2,1,1,0,0,0,0,0],[999,1,1,1,1,1,1,1,1,1,1,1,1,1,1,1,1,1,1,1,1,1],[1,1,1,1,1,1,1,1,1,1,1,1,1,1,1,1,1,1,1,1,1,1],[1,1,1,1,1,1,1,1,1,1,1,1,1,1,1,1,1,1,1,1,1,1],[1,1,1,1,1,1,1,1,1,1,1,1,1,1,1,1,1,1,1,1,1,1],[1,1,1,1,1,1,1,1,1,1,1,1,1,1,1,1,1,1,1,1,1,1],[1,1,1,1,1,1,1,1,1,1,1,1,1,1,1,1,1,1,1,1,1,1]],[[1,0,-2,2,50,0,60,5,36.5,230,360,1,2,2,2,1,1,0,0,0,0,0],[2,0,-2,2,50,0,60,5,36.5,230,360,1,2,2,2,1,1,0,0,0,0,0],[3,0,-2,2,50,0,60,5,36.5,230,360,1,2,2,2,1,1,0,0,0,0,0],[4,0,-2,2,50,0,60,5,36.5,230,360,1,2,2,2,1,1,0,0,0,0,0],[999,1,1,1,1,1,1,1,1,1,1,1,1,1,1,1,1,1,1,1,1,1],[1,1,1,1,1,1,1,1,1,1,1,1,1,1,1,1,1,1,1,1,1,1],[1,1,1,1,1,1,1,1,1,1,1,1,1,1,1,1,1,1,1,1,1,1],[1,1,1,1,1,1,1,1,1,1,1,1,1,1,1,1,1,1,1,1,1,1],[1,1,1,1,1,1,1,1,1,1,1,1,1,1,1,1,1,1,1,1,1,1],[1,1,1,1,1,1,1,1,1,1,1,1,1,1,1,1,1,1,1,1,1,1]]];
    ![[[1,0,-2,2,50,38,60,5,36.5,230,370,1,2,2,2,1,1,0,0,0,0,0],[2,0,-2,2,50,38,60,5,36.5,230,370,1,2,2,2,1,1,0,0,0,0,0],[3,0,-2,2,50,38,60,5,36.5,230,370,1,2,2,2,1,1,0,0,0,0,0],[4,0,-2,2,50,38,60,5,36.5,230,370,1,2,2,2,1,1,0,0,0,0,0],[999,1,1,1,1,1,1,1,1,1,1,1,1,1,1,1,1,1,1,1,1,1],[1,1,1,1,1,1,1,1,1,1,1,1,1,1,1,1,1,1,1,1,1,1],[1,1,1,1,1,1,1,1,1,1,1,1,1,1,1,1,1,1,1,1,1,1],[1,1,1,1,1,1,1,1,1,1,1,1,1,1,1,1,1,1,1,1,1,1],[1,1,1,1,1,1,1,1,1,1,1,1,1,1,1,1,1,1,1,1,1,1],[1,1,1,1,1,1,1,1,1,1,1,1,1,1,1,1,1,1,1,1,1,1]],[[1,0,-2,2,50,38,60,5,36.5,230,360,1,2,2,2,1,1,0,0,0,0,0],[2,0,-2,2,50,38,60,5,36.5,230,360,1,2,2,2,1,1,0,0,0,0,0],[3,0,-2,2,50,38,60,5,36.5,230,360,1,2,2,2,1,1,0,0,0,0,0],[4,0,-2,2,50,38,60,5,36.5,230,360,1,2,2,2,1,1,0,0,0,0,0],[999,1,1,1,1,1,1,1,1,1,1,1,1,1,1,1,1,1,1,1,1,1],[1,1,1,1,1,1,1,1,1,1,1,1,1,1,1,1,1,1,1,1,1,1],[1,1,1,1,1,1,1,1,1,1,1,1,1,1,1,1,1,1,1,1,1,1],[1,1,1,1,1,1,1,1,1,1,1,1,1,1,1,1,1,1,1,1,1,1],[1,1,1,1,1,1,1,1,1,1,1,1,1,1,1,1,1,1,1,1,1,1],[1,1,1,1,1,1,1,1,1,1,1,1,1,1,1,1,1,1,1,1,1,1]]];
    PERS torchmotion macroManualEndA{2,10}:=[[[1,-3,-2,2,50,0,60,5,36.5,230,380,1,2,2,1.5,1,1,0,10,20,30,0],[2,-2,-2,2,50,0,60,5,36.5,230,380,1,2,2,1.5,1,1,0,0,0,0,0],[3,-1,-2,2,50,0,60,5,36.5,230,380,1,2,2,1.5,1,1,0,0,0,0,0],[4,0,-2,2,50,0,60,5,36.5,230,380,1,2,2,1.5,1,1,0,0,0,0,0],[999,1,1,1,1,1,1,1,1,1,1,1,1,1,1,1,1,1,1,1,1,1],[1,1,1,1,1,1,1,1,1,1,1,1,1,1,1,1,1,1,1,1,1,1],[1,1,1,1,1,1,1,1,1,1,1,1,1,1,1,1,1,1,1,1,1,1],[1,1,1,1,1,1,1,1,1,1,1,1,1,1,1,1,1,1,1,1,1,1],[1,1,1,1,1,1,1,1,1,1,1,1,1,1,1,1,1,1,1,1,1,1],[1,1,1,1,1,1,1,1,1,1,1,1,1,1,1,1,1,1,1,1,1,1]],[[1,-3,-3,2,50,0,60,5,36.3,232,360,1,2,2,1.5,1,1,0,10,20,30,0],[2,-2,-3,2,50,0,60,5,36.3,232,360,1,2,2,1.5,1,1,0,0,0,0,0],[3,-1,-2,2,50,0,60,5,36.3,232,360,1,2,2,1.5,1,1,0,0,0,0,0],[4,0,-2,2,50,0,60,5,36.3,232,360,1,2,2,1.5,1,1,0,0,0,0,0],[999,1,1,1,1,1,1,1,1,1,1,1,1,1,1,1,1,1,1,1,1,1],[1,1,1,1,1,1,1,1,1,1,1,1,1,1,1,1,1,1,1,1,1,1],[1,1,1,1,1,1,1,1,1,1,1,1,1,1,1,1,1,1,1,1,1,1],[1,1,1,1,1,1,1,1,1,1,1,1,1,1,1,1,1,1,1,1,1,1],[1,1,1,1,1,1,1,1,1,1,1,1,1,1,1,1,1,1,1,1,1,1],[1,1,1,1,1,1,1,1,1,1,1,1,1,1,1,1,1,1,1,1,1,1]]];
    ![[[1,0,-2,2,50,-38,60,5,36.5,230,370,1,2,2,2,1,1,0,0,0,0,0],[2,0,-2,2,50,-38,60,5,36.5,230,370,1,2,2,2,1,1,0,0,0,0,0],[3,0,-2,2,50,-38,60,5,36.5,230,370,1,2,2,2,1,1,0,0,0,0,0],[4,0,-2,2,50,-38,60,5,36.5,230,370,1,2,2,2,1,1,0,0,0,0,0],[999,1,1,1,1,1,1,1,1,1,1,1,1,1,1,1,1,1,1,1,1,1],[1,1,1,1,1,1,1,1,1,1,1,1,1,1,1,1,1,1,1,1,1,1],[1,1,1,1,1,1,1,1,1,1,1,1,1,1,1,1,1,1,1,1,1,1],[1,1,1,1,1,1,1,1,1,1,1,1,1,1,1,1,1,1,1,1,1,1],[1,1,1,1,1,1,1,1,1,1,1,1,1,1,1,1,1,1,1,1,1,1],[1,1,1,1,1,1,1,1,1,1,1,1,1,1,1,1,1,1,1,1,1,1]],[[1,0,-2,2,50,-38,60,5,36.5,230,360,1,2,2,2,1,1,0,0,0,0,0],[2,0,-2,2,50,-38,60,5,36.5,230,360,1,2,2,2,1,1,0,0,0,0,0],[3,0,-2,2,50,-38,60,5,36.5,230,360,1,2,2,2,1,1,0,0,0,0,0],[4,0,-2,2,50,-38,60,5,36.5,230,360,1,2,2,2,1,1,0,0,0,0,0],[999,1,1,1,1,1,1,1,1,1,1,1,1,1,1,1,1,1,1,1,1,1],[1,1,1,1,1,1,1,1,1,1,1,1,1,1,1,1,1,1,1,1,1,1],[1,1,1,1,1,1,1,1,1,1,1,1,1,1,1,1,1,1,1,1,1,1],[1,1,1,1,1,1,1,1,1,1,1,1,1,1,1,1,1,1,1,1,1,1],[1,1,1,1,1,1,1,1,1,1,1,1,1,1,1,1,1,1,1,1,1,1],[1,1,1,1,1,1,1,1,1,1,1,1,1,1,1,1,1,1,1,1,1,1]]];
    ![[[1,0,-2,2,50,0,60,5,37,230,380,1,2,2,2,1,1,0,0,0,0,0],[2,0,-2,2,50,0,60,5,37,230,380,1,2,2,2,1,1,0,0,0,0,0],[3,0,-2,2,50,0,60,5,37,230,380,1,2,2,2,1,1,0,0,0,0,0],[4,0,-2,2,50,0,60,5,37,230,380,1,2,2,2,1,1,0,0,0,0,0],[999,1,1,1,1,1,1,1,1,1,1,1,1,1,1,1,1,1,1,1,1,1],[1,1,1,1,1,1,1,1,1,1,1,1,1,1,1,1,1,1,1,1,1,1],[1,1,1,1,1,1,1,1,1,1,1,1,1,1,1,1,1,1,1,1,1,1],[1,1,1,1,1,1,1,1,1,1,1,1,1,1,1,1,1,1,1,1,1,1],[1,1,1,1,1,1,1,1,1,1,1,1,1,1,1,1,1,1,1,1,1,1],[1,1,1,1,1,1,1,1,1,1,1,1,1,1,1,1,1,1,1,1,1,1]],[[1,0,-2,2,50,0,60,5,36.5,230,360,1,2,2,2,1,1,0,0,0,0,0],[2,0,-2,2,50,0,60,5,36.5,230,360,1,2,2,2,1,1,0,0,0,0,0],[3,0,-2,2,50,0,60,5,36.5,230,360,1,2,2,2,1,1,0,0,0,0,0],[4,0,-2,2,50,0,60,5,36.5,230,360,1,2,2,2,1,1,0,0,0,0,0],[999,1,1,1,1,1,1,1,1,1,1,1,1,1,1,1,1,1,1,1,1,1],[1,1,1,1,1,1,1,1,1,1,1,1,1,1,1,1,1,1,1,1,1,1],[1,1,1,1,1,1,1,1,1,1,1,1,1,1,1,1,1,1,1,1,1,1],[1,1,1,1,1,1,1,1,1,1,1,1,1,1,1,1,1,1,1,1,1,1],[1,1,1,1,1,1,1,1,1,1,1,1,1,1,1,1,1,1,1,1,1,1],[1,1,1,1,1,1,1,1,1,1,1,1,1,1,1,1,1,1,1,1,1,1]]];
    PERS torchmotion macroManualEndB{2,10}:=[[[1,-3,-2,2,50,0,60,5,36.5,230,380,1,2,2,1.5,1,1,0,10,20,30,0],[2,-2,-2,2,50,0,60,5,36.5,230,380,1,2,2,1.5,1,1,0,0,0,0,0],[3,-1,-2,2,50,0,60,5,36.5,230,380,1,2,2,1.5,1,1,0,0,0,0,0],[4,0,-2,2,50,0,60,5,36.5,230,380,1,2,2,1.5,1,1,0,0,0,0,0],[999,1,1,1,1,1,1,1,1,1,1,1,1,1,1,1,1,1,1,1,1,1],[1,1,1,1,1,1,1,1,1,1,1,1,1,1,1,1,1,1,1,1,1,1],[1,1,1,1,1,1,1,1,1,1,1,1,1,1,1,1,1,1,1,1,1,1],[1,1,1,1,1,1,1,1,1,1,1,1,1,1,1,1,1,1,1,1,1,1],[1,1,1,1,1,1,1,1,1,1,1,1,1,1,1,1,1,1,1,1,1,1],[1,1,1,1,1,1,1,1,1,1,1,1,1,1,1,1,1,1,1,1,1,1]],[[1,-3,-3,2,50,0,60,5,36.3,232,360,1,2,2,1.5,1,1,0,10,20,30,0],[2,-2,-3,2,50,0,60,5,36.3,232,360,1,2,2,1.5,1,1,0,0,0,0,0],[3,-1,-2,2,50,0,60,5,36.3,232,360,1,2,2,1.5,1,1,0,0,0,0,0],[4,0,-2,2,50,0,60,5,36.3,232,360,1,2,2,1.5,1,1,0,0,0,0,0],[999,1,1,1,1,1,1,1,1,1,1,1,1,1,1,1,1,1,1,1,1,1],[1,1,1,1,1,1,1,1,1,1,1,1,1,1,1,1,1,1,1,1,1,1],[1,1,1,1,1,1,1,1,1,1,1,1,1,1,1,1,1,1,1,1,1,1],[1,1,1,1,1,1,1,1,1,1,1,1,1,1,1,1,1,1,1,1,1,1],[1,1,1,1,1,1,1,1,1,1,1,1,1,1,1,1,1,1,1,1,1,1],[1,1,1,1,1,1,1,1,1,1,1,1,1,1,1,1,1,1,1,1,1,1]]];
    ![[[1,0,-2,2,50,0,60,5,37,230,380,1,2,2,2,1,1,0,0,0,0,0],[2,0,-2,2,50,0,60,5,37,230,380,1,2,2,2,1,1,0,0,0,0,0],[3,0,-2,2,50,0,60,5,37,230,380,1,2,2,2,1,1,0,0,0,0,0],[4,0,-2,2,50,0,60,5,37,230,380,1,2,2,2,1,1,0,0,0,0,0],[999,1,1,1,1,1,1,1,1,1,1,1,1,1,1,1,1,1,1,1,1,1],[1,1,1,1,1,1,1,1,1,1,1,1,1,1,1,1,1,1,1,1,1,1],[1,1,1,1,1,1,1,1,1,1,1,1,1,1,1,1,1,1,1,1,1,1],[1,1,1,1,1,1,1,1,1,1,1,1,1,1,1,1,1,1,1,1,1,1],[1,1,1,1,1,1,1,1,1,1,1,1,1,1,1,1,1,1,1,1,1,1],[1,1,1,1,1,1,1,1,1,1,1,1,1,1,1,1,1,1,1,1,1,1]],[[1,0,-2,2,50,0,60,5,36.5,230,360,1,2,2,2,1,1,0,0,0,0,0],[2,0,-2,2,50,0,60,5,36.5,230,360,1,2,2,2,1,1,0,0,0,0,0],[3,0,-2,2,50,0,60,5,36.5,230,360,1,2,2,2,1,1,0,0,0,0,0],[4,0,-2,2,50,0,60,5,36.5,230,360,1,2,2,2,1,1,0,0,0,0,0],[999,1,1,1,1,1,1,1,1,1,1,1,1,1,1,1,1,1,1,1,1,1],[1,1,1,1,1,1,1,1,1,1,1,1,1,1,1,1,1,1,1,1,1,1],[1,1,1,1,1,1,1,1,1,1,1,1,1,1,1,1,1,1,1,1,1,1],[1,1,1,1,1,1,1,1,1,1,1,1,1,1,1,1,1,1,1,1,1,1],[1,1,1,1,1,1,1,1,1,1,1,1,1,1,1,1,1,1,1,1,1,1],[1,1,1,1,1,1,1,1,1,1,1,1,1,1,1,1,1,1,1,1,1,1]]];
    ![[[1,0,-2,2,50,-38,60,5,36.5,230,370,1,2,2,2,1,1,0,0,0,0,0],[2,0,-2,2,50,-38,60,5,36.5,230,370,1,2,2,2,1,1,0,0,0,0,0],[3,0,-2,2,50,-38,60,5,36.5,230,370,1,2,2,2,1,1,0,0,0,0,0],[4,0,-2,2,50,-38,60,5,36.5,230,370,1,2,2,2,1,1,0,0,0,0,0],[999,1,1,1,1,1,1,1,1,1,1,1,1,1,1,1,1,1,1,1,1,1],[1,1,1,1,1,1,1,1,1,1,1,1,1,1,1,1,1,1,1,1,1,1],[1,1,1,1,1,1,1,1,1,1,1,1,1,1,1,1,1,1,1,1,1,1],[1,1,1,1,1,1,1,1,1,1,1,1,1,1,1,1,1,1,1,1,1,1],[1,1,1,1,1,1,1,1,1,1,1,1,1,1,1,1,1,1,1,1,1,1],[1,1,1,1,1,1,1,1,1,1,1,1,1,1,1,1,1,1,1,1,1,1]],[[1,0,-2,2,50,-38,60,5,36.5,230,360,1,2,2,2,1,1,0,0,0,0,0],[2,0,-2,2,50,-38,60,5,36.5,230,360,1,2,2,2,1,1,0,0,0,0,0],[3,0,-2,2,50,-38,60,5,36.5,230,360,1,2,2,2,1,1,0,0,0,0,0],[4,0,-2,2,50,-38,60,5,36.5,230,360,1,2,2,2,1,1,0,0,0,0,0],[999,1,1,1,1,1,1,1,1,1,1,1,1,1,1,1,1,1,1,1,1,1],[1,1,1,1,1,1,1,1,1,1,1,1,1,1,1,1,1,1,1,1,1,1],[1,1,1,1,1,1,1,1,1,1,1,1,1,1,1,1,1,1,1,1,1,1],[1,1,1,1,1,1,1,1,1,1,1,1,1,1,1,1,1,1,1,1,1,1],[1,1,1,1,1,1,1,1,1,1,1,1,1,1,1,1,1,1,1,1,1,1],[1,1,1,1,1,1,1,1,1,1,1,1,1,1,1,1,1,1,1,1,1,1]]];

    PERS torchmotion macroStartBuffer1{10}:=[[1,0,-2,2,50,0,60,5,36.8,230,380,1,2,2,1.5,1,1,0,0,0,0,0],[2,1,-2,2,50,0,60,5,36.8,230,380,1,2,2,1.5,1,1,0,0,0,0,0],[3,2,-2,2,50,0,60,5,36.8,230,380,1,2,2,1.5,1,1,0,0,0,0,0],[4,3,-2,2,50,0,60,5,36.8,230,380,1,2,2,1.5,1,1,0,0,0,0,0],[999,1,1,1,1,1,1,1,1,1,1,1,1,1,1,1,1,1,1,1,1,1],[1,1,1,1,1,1,1,1,1,1,1,1,1,1,1,1,1,1,1,1,1,1],[1,1,1,1,1,1,1,1,1,1,1,1,1,1,1,1,1,1,1,1,1,1],[1,1,1,1,1,1,1,1,1,1,1,1,1,1,1,1,1,1,1,1,1,1],[1,1,1,1,1,1,1,1,1,1,1,1,1,1,1,1,1,1,1,1,1,1],[1,1,1,1,1,1,1,1,1,1,1,1,1,1,1,1,1,1,1,1,1,1]];
    PERS torchmotion macroStartBuffer2{10}:=[[1,0,-3,2,50,0,60,5,36.3,232,360,1,2,2,1.5,1,1,0,0,0,0,0],[2,1,-3,2,50,0,60,5,36.3,232,360,1,2,2,1.5,1,1,0,0,0,0,0],[3,2,-3,2,50,0,60,5,36.3,232,360,1,2,2,1.5,1,1,0,0,0,0,0],[4,3,-3,2,50,0,60,5,36.3,232,360,1,2,2,1.5,1,1,0,0,0,0,0],[999,1,1,1,1,1,1,1,1,1,1,1,1,1,1,1,1,1,1,1,1,1],[1,1,1,1,1,1,1,1,1,1,1,1,1,1,1,1,1,1,1,1,1,1],[1,1,1,1,1,1,1,1,1,1,1,1,1,1,1,1,1,1,1,1,1,1],[1,1,1,1,1,1,1,1,1,1,1,1,1,1,1,1,1,1,1,1,1,1],[1,1,1,1,1,1,1,1,1,1,1,1,1,1,1,1,1,1,1,1,1,1],[1,1,1,1,1,1,1,1,1,1,1,1,1,1,1,1,1,1,1,1,1,1]];
    PERS torchmotion macroEndBuffer1{10}:=[[1,-3,-2,2,50,0,60,5,36.8,230,380,1,2,2,1.5,1,1,0,10,20,30,0],[2,-2,-2,2,50,0,60,5,36.8,230,380,1,2,2,1.5,1,1,0,0,0,0,0],[3,-1,-2,2,50,0,60,5,36.8,230,380,1,2,2,1.5,1,1,0,0,0,0,0],[4,0,-2,2,50,0,60,5,36.8,230,380,1,2,2,1.5,1,1,0,0,0,0,0],[999,1,1,1,1,1,1,1,1,1,1,1,1,1,1,1,1,1,1,1,1,1],[1,1,1,1,1,1,1,1,1,1,1,1,1,1,1,1,1,1,1,1,1,1],[1,1,1,1,1,1,1,1,1,1,1,1,1,1,1,1,1,1,1,1,1,1],[1,1,1,1,1,1,1,1,1,1,1,1,1,1,1,1,1,1,1,1,1,1],[1,1,1,1,1,1,1,1,1,1,1,1,1,1,1,1,1,1,1,1,1,1],[1,1,1,1,1,1,1,1,1,1,1,1,1,1,1,1,1,1,1,1,1,1]];
    PERS torchmotion macroEndBuffer2{10}:=[[1,-3,-3,2,50,0,60,5,36.3,232,360,1,2,2,1.5,1,1,0,10,20,30,0],[2,-2,-3,2,50,0,60,5,36.3,232,360,1,2,2,1.5,1,1,0,0,0,0,0],[3,-1,-2,2,50,0,60,5,36.3,232,360,1,2,2,1.5,1,1,0,0,0,0,0],[4,0,-2,2,50,0,60,5,36.3,232,360,1,2,2,1.5,1,1,0,0,0,0,0],[999,1,1,1,1,1,1,1,1,1,1,1,1,1,1,1,1,1,1,1,1,1],[1,1,1,1,1,1,1,1,1,1,1,1,1,1,1,1,1,1,1,1,1,1],[1,1,1,1,1,1,1,1,1,1,1,1,1,1,1,1,1,1,1,1,1,1],[1,1,1,1,1,1,1,1,1,1,1,1,1,1,1,1,1,1,1,1,1,1],[1,1,1,1,1,1,1,1,1,1,1,1,1,1,1,1,1,1,1,1,1,1],[1,1,1,1,1,1,1,1,1,1,1,1,1,1,1,1,1,1,1,1,1,1]];



    !!! Teaching Pose !!!
    PERS jointtarget jTeachPose10:=[[0,-11.58,-54.61,0,-23.21,0],[9E+09,9E+09,9E+09,9E+09,9E+09,9E+09]];
    PERS jointtarget jTeachPose20:=[[0,-13.77,-51.14,0,-24.5,0],[9E+09,9E+09,9E+09,9E+09,9E+09,9E+09]];
    PERS jointtarget jTeachPose30:=[[0,-5.48,-66.86,0,-35.66,0],[9E+09,9E+09,9E+09,9E+09,9E+09,9E+09]];
    PERS jointtarget jTeachPose40:=[[0,-95,70,0,-35,0],[9E+09,9E+09,9E+09,9E+09,9E+09,9E+09]];

    !!! Wire Cut !!!
    PERS jointtarget jWireCutRdy10:=[[-5.74337,56.5223,-2.36426,0,0,0],[-7805.23,-7805.23,1917.83,1534,9E+09,9E+09]];
    PERS jointtarget jWireCutRdy20:=[[-4.42117,43.9252,29.766,35.9723,-31.0497,-17.7691],[-7805.23,-7805.23,1917.83,1534,9E+09,9E+09]];
    PERS jointtarget jWireCutRdy30:=[[-2.45489,39.2604,46.5236,54.029,-43.8022,-8.52495],[-7805.23,-7805.23,1917.83,1534,9E+09,9E+09]];
    PERS jointtarget jWireCutRdy40:=[[-8.44041,38.4714,56.4802,74.9109,-46.3356,6.60117],[-7805.23,-7805.23,1917.83,1534,9E+09,9E+09]];
    PERS jointtarget jWireCut:=[[-10.3272,38.7931,61.3627,68.3466,-47.9698,13.406],[-7805.23,-7805.23,1917.83,1534,9E+09,9E+09]];
    PERS jointtarget jWireCutRdy50:=[[-8.44041,38.4714,56.4802,74.9108,-46.3356,6.60084],[-7805.23,-7805.23,1917.83,1534,9E+09,9E+09]];
    PERS jointtarget jWireCutRdy60:=[[-4.42128,43.9251,29.766,35.9723,-31.0497,-17.7691],[-7805.23,-7805.23,1917.83,1534,9E+09,9E+09]];
    PERS jointtarget jWireCutRdy70:=[[-5.74337,56.5222,-2.36431,0,0,0],[-7805.23,-7805.23,1917.83,1534,9E+09,9E+09]];

    !!! rNozzle Clean !!!
    PERS jointtarget jNozzleClean10:=[[92.7023,56.7732,-24.6002,-105.292,47.2145,-39.1763],[-7.83472,-7.83523,5212.01,422.601,9E+09,9E+09]];
    PERS jointtarget jNozzleClean20:=[[154.238,56.7746,-24.5971,-105.291,47.2139,-39.1774],[-7.83472,-7.83495,5212.01,422.595,9E+09,9E+09]];
    PERS jointtarget jNozzleClean30:=[[144.266,78.8984,-24.7284,-105.291,47.2139,-39.1774],[-7.83513,-7.83495,5212.01,422.596,9E+09,9E+09]];
    PERS jointtarget jNozzleClean40:=[[136.493,90.5978,-51.7581,-95.8271,39.0251,-59.7871],[-7.83513,-7.83482,5212.01,422.595,9E+09,9E+09]];
    PERS jointtarget jNozzleClean:=[[136.493,90.5979,-51.7581,-95.8269,39.0251,-59.7873],[-7.83513,-7.83495,5212.01,422.595,9E+09,9E+09]];
    PERS jointtarget jNozzleClean50:=[[136.493,90.5979,-51.7581,-95.8269,39.0252,-59.7873],[-7.83513,-7.83495,5212.01,422.595,9E+09,9E+09]];
    PERS jointtarget jNozzleClean60:=[[144.266,78.8983,-24.7285,-105.291,47.2139,-39.1774],[-7.83513,-7.83495,5212.01,422.595,9E+09,9E+09]];
    PERS jointtarget jNozzleClean70:=[[154.238,56.7746,-24.5971,-105.291,47.2139,-39.1774],[-7.83513,-7.83495,5212.01,422.595,9E+09,9E+09]];
    PERS jointtarget jNozzleClean80:=[[92.7023,56.7732,-24.6003,-105.292,47.2145,-39.176],[-7.83472,-7.83523,5212.01,422.601,9E+09,9E+09]];

    PERS jointgroup ManualOrigin_Pos:=[[[90,90,-45,0,20,0],[9E+09,9E+09,9E+09,9E+09,9E+09,9E+09]],[[90,90,-45,0,20,0],[9E+09,9E+09,9E+09,9E+09,9E+09,9E+09]],[[9E+09,9E+09,9E+09,9E+09,9E+09,9E+09],[1391,5300,841,0,9E+09,1391]]];

    PERS robtarget pWeldPosR1{40}:=[[[-3,7,1],[0.307623,-0.549545,-0.742667,-0.227629],[-1,0,0,1],[-8704.03,-8704.03,294.161,1030.31,9E+9,9E+9]],[[-3,7,1],[0.307623,-0.549545,-0.742667,-0.227629],[-1,0,0,1],[-8704.03,-8704.03,294.161,1030.31,9E+9,9E+9]],[[-3,-4.5,1],[0.307623,-0.549545,-0.742667,-0.227629],[-1,0,0,1],[-8704.03,-8704.03,294.161,1030.31,9E+9,9E+9]],[[15,-1,1],[0.307623,-0.549545,-0.742667,-0.227629],[-1,0,0,1],[-8704.03,-8704.03,294.161,1030.34,9E+9,9E+9]],[[200,-1,1],[0.270598,-0.653282,-0.653282,-0.270598],[-1,0,0,1],[-8704.03,-8704.03,294.161,1030.72,9E+9,9E+9]],[[1390,-1.00592,0.996463],[0.270597,-0.653283,-0.653281,-0.270597],[0,0,-1,1],[-8707.81,-8707.8,1477.15,1033.13,9E+9,9E+9]],[[0,0,0],[0,0,0,0],[0,0,0,0],[0,0,0,0,0,0]],[[0,0,0],[0,0,0,0],[0,0,0,0],[0,0,0,0,0,0]],[[0,0,0],[0,0,0,0],[0,0,0,0],[0,0,0,0,0,0]],[[0,0,0],[0,0,0,0],[0,0,0,0],[0,0,0,0,0,0]],[[0,0,0],[0,0,0,0],[0,0,0,0],[0,0,0,0,0,0]],[[0,0,0],[0,0,0,0],[0,0,0,0],[0,0,0,0,0,0]],[[0,0,0],[0,0,0,0],[0,0,0,0],[0,0,0,0,0,0]],[[0,0,0],[0,0,0,0],[0,0,0,0],[0,0,0,0,0,0]],[[0,0,0],[0,0,0,0],[0,0,0,0],[0,0,0,0,0,0]],[[0,0,0],[0,0,0,0],[0,0,0,0],[0,0,0,0,0,0]],[[0,0,0],[0,0,0,0],[0,0,0,0],[0,0,0,0,0,0]],[[0,0,0],[0,0,0,0],[0,0,0,0],[0,0,0,0,0,0]],[[0,0,0],[0,0,0,0],[0,0,0,0],[0,0,0,0,0,0]],[[0,0,0],[0,0,0,0],[0,0,0,0],[0,0,0,0,0,0]],[[0,0,0],[0,0,0,0],[0,0,0,0],[0,0,0,0,0,0]],[[0,0,0],[0,0,0,0],[0,0,0,0],[0,0,0,0,0,0]],[[0,0,0],[0,0,0,0],[0,0,0,0],[0,0,0,0,0,0]],[[0,0,0],[0,0,0,0],[0,0,0,0],[0,0,0,0,0,0]],[[0,0,0],[0,0,0,0],[0,0,0,0],[0,0,0,0,0,0]],[[0,0,0],[0,0,0,0],[0,0,0,0],[0,0,0,0,0,0]],[[0,0,0],[0,0,0,0],[0,0,0,0],[0,0,0,0,0,0]],[[0,0,0],[0,0,0,0],[0,0,0,0],[0,0,0,0,0,0]],[[0,0,0],[0,0,0,0],[0,0,0,0],[0,0,0,0,0,0]],[[0,0,0],[0,0,0,0],[0,0,0,0],[0,0,0,0,0,0]],[[0,0,0],[0,0,0,0],[0,0,0,0],[0,0,0,0,0,0]],[[0,0,0],[0,0,0,0],[0,0,0,0],[0,0,0,0,0,0]],[[0,0,0],[0,0,0,0],[0,0,0,0],[0,0,0,0,0,0]],[[0,0,0],[0,0,0,0],[0,0,0,0],[0,0,0,0,0,0]],[[0,0,0],[0,0,0,0],[0,0,0,0],[0,0,0,0,0,0]],[[0,0,0],[0,0,0,0],[0,0,0,0],[0,0,0,0,0,0]],[[0,0,0],[0,0,0,0],[0,0,0,0],[0,0,0,0,0,0]],[[0,0,0],[0,0,0,0],[0,0,0,0],[0,0,0,0,0,0]],[[0,0,0],[0,0,0,0],[0,0,0,0],[0,0,0,0,0,0]],[[15,-1,1],[0.307623,-0.549545,-0.742667,-0.227629],[-1,0,0,1],[-8704.03,-8704.03,294.161,1030.34,9E+9,9E+9]]];
    PERS robtarget pWeldPosR2{40}:=[[[-3,7,1],[0.307623,-0.549545,-0.742667,-0.227629],[-1,0,0,1],[-8704.03,-8704.03,294.161,1030.31,9E+09,9E+09]],[[-3,7,1],[0.307623,-0.549545,-0.742667,-0.227629],[-1,0,0,1],[-8704.03,-8704.03,294.161,1030.31,9E+09,9E+09]],[[-3,-4.5,1],[0.307623,-0.549545,-0.742667,-0.227629],[-1,0,0,1],[-8704.03,-8704.03,294.161,1030.31,9E+09,9E+09]],[[15,-1,1],[0.307623,-0.549545,-0.742667,-0.227629],[-1,0,0,1],[-8704.03,-8704.03,294.161,1030.34,9E+09,9E+09]],[[200,-1,1],[0.270598,-0.653282,-0.653282,-0.270598],[-1,0,0,1],[-8704.03,-8704.03,294.161,1030.72,9E+09,9E+09]],[[1390,-1.00592,0.996463],[0.270597,-0.653283,-0.653281,-0.270597],[0,0,-1,1],[-8707.81,-8707.8,1477.15,1033.13,9E+09,9E+09]],[[0,0,0],[0,0,0,0],[0,0,0,0],[0,0,0,0,0,0]],[[0,0,0],[0,0,0,0],[0,0,0,0],[0,0,0,0,0,0]],[[0,0,0],[0,0,0,0],[0,0,0,0],[0,0,0,0,0,0]],[[0,0,0],[0,0,0,0],[0,0,0,0],[0,0,0,0,0,0]],[[0,0,0],[0,0,0,0],[0,0,0,0],[0,0,0,0,0,0]],[[0,0,0],[0,0,0,0],[0,0,0,0],[0,0,0,0,0,0]],[[0,0,0],[0,0,0,0],[0,0,0,0],[0,0,0,0,0,0]],[[0,0,0],[0,0,0,0],[0,0,0,0],[0,0,0,0,0,0]],[[0,0,0],[0,0,0,0],[0,0,0,0],[0,0,0,0,0,0]],[[0,0,0],[0,0,0,0],[0,0,0,0],[0,0,0,0,0,0]],[[0,0,0],[0,0,0,0],[0,0,0,0],[0,0,0,0,0,0]],[[0,0,0],[0,0,0,0],[0,0,0,0],[0,0,0,0,0,0]],[[0,0,0],[0,0,0,0],[0,0,0,0],[0,0,0,0,0,0]],[[0,0,0],[0,0,0,0],[0,0,0,0],[0,0,0,0,0,0]],[[0,0,0],[0,0,0,0],[0,0,0,0],[0,0,0,0,0,0]],[[0,0,0],[0,0,0,0],[0,0,0,0],[0,0,0,0,0,0]],[[0,0,0],[0,0,0,0],[0,0,0,0],[0,0,0,0,0,0]],[[0,0,0],[0,0,0,0],[0,0,0,0],[0,0,0,0,0,0]],[[0,0,0],[0,0,0,0],[0,0,0,0],[0,0,0,0,0,0]],[[0,0,0],[0,0,0,0],[0,0,0,0],[0,0,0,0,0,0]],[[0,0,0],[0,0,0,0],[0,0,0,0],[0,0,0,0,0,0]],[[0,0,0],[0,0,0,0],[0,0,0,0],[0,0,0,0,0,0]],[[0,0,0],[0,0,0,0],[0,0,0,0],[0,0,0,0,0,0]],[[0,0,0],[0,0,0,0],[0,0,0,0],[0,0,0,0,0,0]],[[0,0,0],[0,0,0,0],[0,0,0,0],[0,0,0,0,0,0]],[[0,0,0],[0,0,0,0],[0,0,0,0],[0,0,0,0,0,0]],[[0,0,0],[0,0,0,0],[0,0,0,0],[0,0,0,0,0,0]],[[0,0,0],[0,0,0,0],[0,0,0,0],[0,0,0,0,0,0]],[[0,0,0],[0,0,0,0],[0,0,0,0],[0,0,0,0,0,0]],[[0,0,0],[0,0,0,0],[0,0,0,0],[0,0,0,0,0,0]],[[0,0,0],[0,0,0,0],[0,0,0,0],[0,0,0,0,0,0]],[[0,0,0],[0,0,0,0],[0,0,0,0],[0,0,0,0,0,0]],[[0,0,0],[0,0,0,0],[0,0,0,0],[0,0,0,0,0,0]],[[1390,-1,1],[0.270598,-0.653282,-0.653282,-0.270598],[-1,0,0,1],[-8707.8,-8707.8,1477.15,1033.12,9E+09,9E+09]]];
    PERS robtarget pWeldPosG{40};
    PERS speeddata vWeld1{40}:=[[10,200,200,200],[10,200,200,200],[10,200,200,200],[10,200,200,200],[10,200,200,200],[10,200,200,200],[0,0,0,0],[0,0,0,0],[0,0,0,0],[0,0,0,0],[0,0,0,0],[0,0,0,0],[0,0,0,0],[0,0,0,0],[0,0,0,0],[0,0,0,0],[0,0,0,0],[0,0,0,0],[0,0,0,0],[0,0,0,0],[0,0,0,0],[0,0,0,0],[0,0,0,0],[0,0,0,0],[0,0,0,0],[0,0,0,0],[0,0,0,0],[0,0,0,0],[0,0,0,0],[0,0,0,0],[0,0,0,0],[0,0,0,0],[0,0,0,0],[0,0,0,0],[0,0,0,0],[0,0,0,0],[0,0,0,0],[0,0,0,0],[0,0,0,0],[10,200,200,200]];
    PERS speeddata vWeld2{40}:=[[10,200,200,200],[10,200,200,200],[10,200,200,200],[10,200,200,200],[10,200,200,200],[10,200,200,200],[0,0,0,0],[0,0,0,0],[0,0,0,0],[0,0,0,0],[0,0,0,0],[0,0,0,0],[0,0,0,0],[0,0,0,0],[0,0,0,0],[0,0,0,0],[0,0,0,0],[0,0,0,0],[0,0,0,0],[0,0,0,0],[0,0,0,0],[0,0,0,0],[0,0,0,0],[0,0,0,0],[0,0,0,0],[0,0,0,0],[0,0,0,0],[0,0,0,0],[0,0,0,0],[0,0,0,0],[0,0,0,0],[0,0,0,0],[0,0,0,0],[0,0,0,0],[0,0,0,0],[0,0,0,0],[0,0,0,0],[0,0,0,0],[0,0,0,0],[10,200,200,200]];

    !!! Speed Data !!!
    PERS speeddata vTargetSpeed:=[400,300,400,25];
    PERS speeddata vTargetSpeed2:=[9,200,200,25];
    PERS speeddata vWeldEntry:=[100,20,200,25];

    !!! variables for Speed Data !!!
    PERS num nWireCutSpeed:=500;
    PERS num nGantrySpeed:=0;
    PERS num nDryRunSpeed:=2.5;

    !!! Zone Data !!!
    PERS zonedata zTargetZone:=[FALSE,30,5,5,2,1,1];
    PERS zonedata zFineZone:=[TRUE,0,0,0,0,0,0];

    VAR num rotationMaxtrix{3,3};

    ! MoveStepGantryHeight
    PERS num nCurrentGantryHeight:=0;
    PERS num nTargetGantryHeight:=-35.9858;
    PERS num nCalculatedGantryHeight:=0;
    PERS num nGantrySafetyHeight:=-100;
    PERS jointtarget jReadyGantryHeightBuffer:=[[9E+09,9E+09,9E+09,9E+09,9E+09,9E+09],[10404,5130.4,-0.000881434,89.8303,9E+09,10404]];
    PERS num nAngleOfEntry:=0.155838;
    PERS num nAngleRzStore:=-89.8299;
    PERS num nCalculatedHeight:=461.831;

    !!! weld data !!!
    TASK PERS welddata wdArray{40}:=[[10,0,[5,0,36.8,230,0,0,0,0,0],[0,0,0,0,0,0,0,0,0]],[10,0,[5,0,36.8,230,0,0,0,0,0],[0,0,0,0,0,0,0,0,0]],[10,0,[5,0,36.8,230,0,0,0,0,0],[0,0,0,0,0,0,0,0,0]],[10,0,[5,0,36.8,230,0,0,0,0,0],[0,0,0,0,0,0,0,0,0]],[10,0,[5,0,36.8,230,0,0,0,0,0],[0,0,0,0,0,0,0,0,0]],[10,0,[5,0,36.8,230,0,0,0,0,0],[0,0,0,0,0,0,0,0,0]],[10,0,[5,0,36.8,230,0,0,0,0,0],[0,0,0,0,0,0,0,0,0]],[10,0,[5,0,36.8,230,0,0,0,0,0],[0,0,0,0,0,0,0,0,0]],[10,0,[5,0,36.8,230,0,0,0,0,0],[0,0,0,0,0,0,0,0,0]],[10,0,[5,0,36.8,230,0,0,0,0,0],[0,0,0,0,0,0,0,0,0]],[10,0,[5,0,34,210,0,0,0,0,0],[0,0,0,0,0,0,0,0,0]],[10,0,[5,0,34,210,0,0,0,0,0],[0,0,0,0,0,0,0,0,0]],[10,0,[5,0,37.5,270,0,0,0,0,0],[0,0,0,0,0,0,0,0,0]],[10,0,[5,0,37.5,250,0,0,0,0,0],[0,0,0,0,0,0,0,0,0]],[10,0,[5,0,37.5,250,0,0,0,0,0],[0,0,0,0,0,0,0,0,0]],[10,0,[5,0,37.5,250,0,0,0,0,0],[0,0,0,0,0,0,0,0,0]],[10,0,[5,0,37.5,250,0,0,0,0,0],[0,0,0,0,0,0,0,0,0]],[10,0,[5,0,37.5,250,0,0,0,0,0],[0,0,0,0,0,0,0,0,0]],[10,0,[5,0,37.5,250,0,0,0,0,0],[0,0,0,0,0,0,0,0,0]],[10,0,[5,0,37.5,250,0,0,0,0,0],[0,0,0,0,0,0,0,0,0]],[0,0,[0,0,0,0,0,0,0,0,0],[0,0,0,0,0,0,0,0,0]],[0,0,[0,0,0,0,0,0,0,0,0],[0,0,0,0,0,0,0,0,0]],[0,0,[0,0,0,0,0,0,0,0,0],[0,0,0,0,0,0,0,0,0]],[0,0,[0,0,0,0,0,0,0,0,0],[0,0,0,0,0,0,0,0,0]],[0,0,[0,0,0,0,0,0,0,0,0],[0,0,0,0,0,0,0,0,0]],[0,0,[0,0,0,0,0,0,0,0,0],[0,0,0,0,0,0,0,0,0]],[0,0,[0,0,0,0,0,0,0,0,0],[0,0,0,0,0,0,0,0,0]],[0,0,[0,0,0,0,0,0,0,0,0],[0,0,0,0,0,0,0,0,0]],[0,0,[0,0,0,0,0,0,0,0,0],[0,0,0,0,0,0,0,0,0]],[0,0,[0,0,0,0,0,0,0,0,0],[0,0,0,0,0,0,0,0,0]],[9,0,[5,0,28,160,0,0,0,0,0],[0,0,0,0,0,0,0,0,0]],[9,0,[5,0,28,160,0,0,0,0,0],[0,0,0,0,0,0,0,0,0]],[9,0,[5,0,28,160,0,0,0,0,0],[0,0,0,0,0,0,0,0,0]],[9,0,[5,0,28,160,0,0,0,0,0],[0,0,0,0,0,0,0,0,0]],[9,0,[5,0,28,160,0,0,0,0,0],[0,0,0,0,0,0,0,0,0]],[9,0,[5,0,28,160,0,0,0,0,0],[0,0,0,0,0,0,0,0,0]],[9,0,[5,0,28,160,0,0,0,0,0],[0,0,0,0,0,0,0,0,0]],[9,0,[5,0,28,160,0,0,0,0,0],[0,0,0,0,0,0,0,0,0]],[9,0,[5,0,28,160,0,0,0,0,0],[0,0,0,0,0,0,0,0,0]],[9,0,[5,0,28,160,0,0,0,0,0],[0,0,0,0,0,0,0,0,0]]];
    TASK PERS welddata wd1:=[10,0,[5,0,36.5,230,0,380,0,0,0],[0,0,0,0,0,0,0,0,0]];
    TASK PERS welddata wd2:=[10,0,[5,0,36.5,230,0,380,0,0,0],[0,0,0,0,0,0,0,0,0]];
    TASK PERS welddata wd3:=[10,0,[5,0,36.5,230,0,380,0,0,0],[0,0,0,0,0,0,0,0,0]];
    TASK PERS welddata wd4:=[10,0,[5,0,36.5,230,0,380,0,0,0],[0,0,0,0,0,0,0,0,0]];
    TASK PERS welddata wd5:=[0,0,[5,0,0,0,0,0,0,0,0],[0,0,0,0,0,0,0,0,0]];
    TASK PERS welddata wd6:=[0,0,[5,0,0,0,0,0,0,0,0],[0,0,0,0,0,0,0,0,0]];
    TASK PERS welddata wd7:=[0,0,[5,0,0,0,0,0,0,0,0],[0,0,0,0,0,0,0,0,0]];
    TASK PERS welddata wd8:=[0,0,[5,0,0,0,0,0,0,0,0],[0,0,0,0,0,0,0,0,0]];
    TASK PERS welddata wd9:=[0,0,[5,0,0,0,0,0,0,0,0],[0,0,0,0,0,0,0,0,0]];
    TASK PERS welddata wd10:=[0,0,[5,0,0,0,0,0,0,0,0],[0,0,0,0,0,0,0,0,0]];
    TASK PERS welddata wd11:=[0,0,[5,0,0,0,0,0,0,0,0],[0,0,0,0,0,0,0,0,0]];
    TASK PERS welddata wd12:=[0,0,[5,0,0,0,0,0,0,0,0],[0,0,0,0,0,0,0,0,0]];
    TASK PERS welddata wd13:=[0,0,[5,0,0,0,0,0,0,0,0],[0,0,0,0,0,0,0,0,0]];
    TASK PERS welddata wd14:=[0,0,[5,0,0,0,0,0,0,0,0],[0,0,0,0,0,0,0,0,0]];
    TASK PERS welddata wd15:=[0,0,[5,0,0,0,0,0,0,0,0],[0,0,0,0,0,0,0,0,0]];
    TASK PERS welddata wd16:=[0,0,[5,0,0,0,0,0,0,0,0],[0,0,0,0,0,0,0,0,0]];
    TASK PERS welddata wd17:=[0,0,[5,0,0,0,0,0,0,0,0],[0,0,0,0,0,0,0,0,0]];
    TASK PERS welddata wd18:=[0,0,[5,0,0,0,0,0,0,0,0],[0,0,0,0,0,0,0,0,0]];
    TASK PERS welddata wd19:=[0,0,[5,0,0,0,0,0,0,0,0],[0,0,0,0,0,0,0,0,0]];
    TASK PERS welddata wd20:=[0,0,[5,0,0,0,0,0,0,0,0],[0,0,0,0,0,0,0,0,0]];
    TASK PERS welddata wd21:=[0,0,[5,0,0,0,0,0,0,0,0],[0,0,0,0,0,0,0,0,0]];
    TASK PERS welddata wd22:=[0,0,[5,0,0,0,0,0,0,0,0],[0,0,0,0,0,0,0,0,0]];
    TASK PERS welddata wd23:=[0,0,[5,0,0,0,0,0,0,0,0],[0,0,0,0,0,0,0,0,0]];
    TASK PERS welddata wd24:=[0,0,[5,0,0,0,0,0,0,0,0],[0,0,0,0,0,0,0,0,0]];
    TASK PERS welddata wd25:=[0,0,[5,0,0,0,0,0,0,0,0],[0,0,0,0,0,0,0,0,0]];
    TASK PERS welddata wd26:=[0,0,[5,0,0,0,0,0,0,0,0],[0,0,0,0,0,0,0,0,0]];
    TASK PERS welddata wd27:=[0,0,[5,0,0,0,0,0,0,0,0],[0,0,0,0,0,0,0,0,0]];
    TASK PERS welddata wd28:=[0,0,[5,0,0,0,0,0,0,0,0],[0,0,0,0,0,0,0,0,0]];
    TASK PERS welddata wd29:=[0,0,[5,0,0,0,0,0,0,0,0],[0,0,0,0,0,0,0,0,0]];
    TASK PERS welddata wd30:=[0,0,[5,0,0,0,0,0,0,0,0],[0,0,0,0,0,0,0,0,0]];
    TASK PERS welddata wd31:=[0,0,[5,0,0,0,0,0,0,0,0],[0,0,0,0,0,0,0,0,0]];
    TASK PERS welddata wd32:=[0,0,[5,0,0,0,0,0,0,0,0],[0,0,0,0,0,0,0,0,0]];
    TASK PERS welddata wd33:=[0,0,[5,0,0,0,0,0,0,0,0],[0,0,0,0,0,0,0,0,0]];
    TASK PERS welddata wd34:=[0,0,[5,0,0,0,0,0,0,0,0],[0,0,0,0,0,0,0,0,0]];
    TASK PERS welddata wd35:=[0,0,[5,0,0,0,0,0,0,0,0],[0,0,0,0,0,0,0,0,0]];
    TASK PERS welddata wd36:=[0,0,[5,0,0,0,0,0,0,0,0],[0,0,0,0,0,0,0,0,0]];
    TASK PERS welddata wd37:=[0,0,[5,0,0,0,0,0,0,0,0],[0,0,0,0,0,0,0,0,0]];
    TASK PERS welddata wd38:=[0,0,[5,0,0,0,0,0,0,0,0],[0,0,0,0,0,0,0,0,0]];
    TASK PERS welddata wd39:=[0,0,[5,0,0,0,0,0,0,0,0],[0,0,0,0,0,0,0,0,0]];
    TASK PERS welddata wd40:=[10,0,[5,0,36.5,230,0,380,0,0,0],[0,0,0,0,0,0,0,0,0]];

    !!! weave data !!!
    TASK PERS weavedata weave1:=[1,2,2.5,1.7,0,0,0,0,0,0,0,0,0,0,0];
    TASK PERS weavedata weave2:=[1,2,2.5,1.7,0,0,0,0,0,0,0,0,0,0,0];
    TASK PERS weavedata weave3:=[1,2,2.5,1.7,0,0,0,0,0,0,0,0,0,0,0];
    TASK PERS weavedata weave4:=[1,2,2.5,1.7,0,0,0,0,0,0,0,0,0,0,0];
    TASK PERS weavedata weave5:=[0,0,0,0,0,0,0,0,0,0,0,0,0,0,0];
    TASK PERS weavedata weave6:=[0,0,0,0,0,0,0,0,0,0,0,0,0,0,0];
    TASK PERS weavedata weave7:=[0,0,0,0,0,0,0,0,0,0,0,0,0,0,0];
    TASK PERS weavedata weave8:=[0,0,0,0,0,0,0,0,0,0,0,0,0,0,0];
    TASK PERS weavedata weave9:=[0,0,0,0,0,0,0,0,0,0,0,0,0,0,0];
    TASK PERS weavedata weave10:=[0,0,0,0,0,0,0,0,0,0,0,0,0,0,0];
    TASK PERS weavedata weave11:=[0,0,0,0,0,0,0,0,0,0,0,0,0,0,0];
    TASK PERS weavedata weave12:=[0,0,0,0,0,0,0,0,0,0,0,0,0,0,0];
    TASK PERS weavedata weave13:=[0,0,0,0,0,0,0,0,0,0,0,0,0,0,0];
    TASK PERS weavedata weave14:=[0,0,0,0,0,0,0,0,0,0,0,0,0,0,0];
    TASK PERS weavedata weave15:=[0,0,0,0,0,0,0,0,0,0,0,0,0,0,0];
    TASK PERS weavedata weave16:=[0,0,0,0,0,0,0,0,0,0,0,0,0,0,0];
    TASK PERS weavedata weave17:=[0,0,0,0,0,0,0,0,0,0,0,0,0,0,0];
    TASK PERS weavedata weave18:=[0,0,0,0,0,0,0,0,0,0,0,0,0,0,0];
    TASK PERS weavedata weave19:=[0,0,0,0,0,0,0,0,0,0,0,0,0,0,0];
    TASK PERS weavedata weave20:=[0,0,0,0,0,0,0,0,0,0,0,0,0,0,0];
    TASK PERS weavedata weave21:=[0,0,0,0,0,0,0,0,0,0,0,0,0,0,0];
    TASK PERS weavedata weave22:=[0,0,0,0,0,0,0,0,0,0,0,0,0,0,0];
    TASK PERS weavedata weave23:=[0,0,0,0,0,0,0,0,0,0,0,0,0,0,0];
    TASK PERS weavedata weave24:=[0,0,0,0,0,0,0,0,0,0,0,0,0,0,0];
    TASK PERS weavedata weave25:=[0,0,0,0,0,0,0,0,0,0,0,0,0,0,0];
    TASK PERS weavedata weave26:=[0,0,0,0,0,0,0,0,0,0,0,0,0,0,0];
    TASK PERS weavedata weave27:=[0,0,0,0,0,0,0,0,0,0,0,0,0,0,0];
    TASK PERS weavedata weave28:=[0,0,0,0,0,0,0,0,0,0,0,0,0,0,0];
    TASK PERS weavedata weave29:=[0,0,0,0,0,0,0,0,0,0,0,0,0,0,0];
    TASK PERS weavedata weave30:=[0,0,0,0,0,0,0,0,0,0,0,0,0,0,0];
    TASK PERS weavedata weave31:=[0,0,0,0,0,0,0,0,0,0,0,0,0,0,0];
    TASK PERS weavedata weave32:=[0,0,0,0,0,0,0,0,0,0,0,0,0,0,0];
    TASK PERS weavedata weave33:=[0,0,0,0,0,0,0,0,0,0,0,0,0,0,0];
    TASK PERS weavedata weave34:=[0,0,0,0,0,0,0,0,0,0,0,0,0,0,0];
    TASK PERS weavedata weave35:=[0,0,0,0,0,0,0,0,0,0,0,0,0,0,0];
    TASK PERS weavedata weave36:=[0,0,0,0,0,0,0,0,0,0,0,0,0,0,0];
    TASK PERS weavedata weave37:=[0,0,0,0,0,0,0,0,0,0,0,0,0,0,0];
    TASK PERS weavedata weave38:=[0,0,0,0,0,0,0,0,0,0,0,0,0,0,0];
    TASK PERS weavedata weave39:=[0,0,0,0,0,0,0,0,0,0,0,0,0,0,0];
    TASK PERS weavedata weave40:=[1,2,2.5,1.7,0,0,0,0,0,0,0,0,0,0,0];

    !!! Track Data !!!
    TASK PERS trackdata track0:=[0,FALSE,50,[0,0,0,0,0,0,0,0,0],[0,0,0,0,0,0,0]];
    TASK PERS trackdata track1:=[0,FALSE,50,[0,15,30,0,0,0,0,0,0],[0,0,0,0,0,0,0]];
    TASK PERS trackdata track2:=[0,FALSE,50,[0,15,30,0,0,0,0,0,0],[0,0,0,0,0,0,0]];
    TASK PERS trackdata track3:=[0,FALSE,50,[0,15,30,0,0,0,0,0,0],[0,0,0,0,0,0,0]];
    TASK PERS trackdata track4:=[0,FALSE,50,[0,15,30,0,0,0,0,0,0],[0,0,0,0,0,0,0]];
    TASK PERS trackdata track5:=[0,FALSE,50,[0,0,0,0,0,0,0,0,0],[0,0,0,0,0,0,0]];
    TASK PERS trackdata track6:=[0,FALSE,50,[0,0,0,0,0,0,0,0,0],[0,0,0,0,0,0,0]];
    TASK PERS trackdata track7:=[0,FALSE,50,[0,0,0,0,0,0,0,0,0],[0,0,0,0,0,0,0]];
    TASK PERS trackdata track8:=[0,FALSE,50,[0,0,0,0,0,0,0,0,0],[0,0,0,0,0,0,0]];
    TASK PERS trackdata track9:=[0,FALSE,50,[0,0,0,0,0,0,0,0,0],[0,0,0,0,0,0,0]];
    TASK PERS trackdata track10:=[0,FALSE,50,[0,0,0,0,0,0,0,0,0],[0,0,0,0,0,0,0]];
    TASK PERS trackdata track11:=[0,FALSE,50,[0,0,0,0,0,0,0,0,0],[0,0,0,0,0,0,0]];
    TASK PERS trackdata track12:=[0,FALSE,50,[0,0,0,0,0,0,0,0,0],[0,0,0,0,0,0,0]];
    TASK PERS trackdata track13:=[0,FALSE,50,[0,0,0,0,0,0,0,0,0],[0,0,0,0,0,0,0]];
    TASK PERS trackdata track14:=[0,FALSE,50,[0,0,0,0,0,0,0,0,0],[0,0,0,0,0,0,0]];
    TASK PERS trackdata track15:=[0,FALSE,50,[0,0,0,0,0,0,0,0,0],[0,0,0,0,0,0,0]];
    TASK PERS trackdata track16:=[0,FALSE,50,[0,0,0,0,0,0,0,0,0],[0,0,0,0,0,0,0]];
    TASK PERS trackdata track17:=[0,FALSE,50,[0,0,0,0,0,0,0,0,0],[0,0,0,0,0,0,0]];
    TASK PERS trackdata track18:=[0,FALSE,50,[0,0,0,0,0,0,0,0,0],[0,0,0,0,0,0,0]];
    TASK PERS trackdata track19:=[0,FALSE,50,[0,0,0,0,0,0,0,0,0],[0,0,0,0,0,0,0]];
    TASK PERS trackdata track20:=[0,FALSE,50,[0,0,0,0,0,0,0,0,0],[0,0,0,0,0,0,0]];
    TASK PERS trackdata track21:=[0,FALSE,50,[0,0,0,0,0,0,0,0,0],[0,0,0,0,0,0,0]];
    TASK PERS trackdata track22:=[0,FALSE,50,[0,0,0,0,0,0,0,0,0],[0,0,0,0,0,0,0]];
    TASK PERS trackdata track23:=[0,FALSE,50,[0,0,0,0,0,0,0,0,0],[0,0,0,0,0,0,0]];
    TASK PERS trackdata track24:=[0,FALSE,50,[0,0,0,0,0,0,0,0,0],[0,0,0,0,0,0,0]];
    TASK PERS trackdata track25:=[0,FALSE,50,[0,0,0,0,0,0,0,0,0],[0,0,0,0,0,0,0]];
    TASK PERS trackdata track26:=[0,FALSE,50,[0,0,0,0,0,0,0,0,0],[0,0,0,0,0,0,0]];
    TASK PERS trackdata track27:=[0,FALSE,50,[0,0,0,0,0,0,0,0,0],[0,0,0,0,0,0,0]];
    TASK PERS trackdata track28:=[0,FALSE,50,[0,0,0,0,0,0,0,0,0],[0,0,0,0,0,0,0]];
    TASK PERS trackdata track29:=[0,FALSE,50,[0,0,0,0,0,0,0,0,0],[0,0,0,0,0,0,0]];
    TASK PERS trackdata track30:=[0,FALSE,50,[0,0,0,0,0,0,0,0,0],[0,0,0,0,0,0,0]];
    TASK PERS trackdata track31:=[0,FALSE,50,[0,0,0,0,0,0,0,0,0],[0,0,0,0,0,0,0]];
    TASK PERS trackdata track32:=[0,FALSE,50,[0,0,0,0,0,0,0,0,0],[0,0,0,0,0,0,0]];
    TASK PERS trackdata track33:=[0,FALSE,50,[0,0,0,0,0,0,0,0,0],[0,0,0,0,0,0,0]];
    TASK PERS trackdata track34:=[0,FALSE,50,[0,0,0,0,0,0,0,0,0],[0,0,0,0,0,0,0]];
    TASK PERS trackdata track35:=[0,FALSE,50,[0,0,0,0,0,0,0,0,0],[0,0,0,0,0,0,0]];
    TASK PERS trackdata track36:=[0,FALSE,50,[0,0,0,0,0,0,0,0,0],[0,0,0,0,0,0,0]];
    TASK PERS trackdata track37:=[0,FALSE,50,[0,0,0,0,0,0,0,0,0],[0,0,0,0,0,0,0]];
    TASK PERS trackdata track38:=[0,FALSE,50,[0,0,0,0,0,0,0,0,0],[0,0,0,0,0,0,0]];
    TASK PERS trackdata track39:=[0,FALSE,50,[0,0,0,0,0,0,0,0,0],[0,0,0,0,0,0,0]];
    TASK PERS trackdata track40:=[0,FALSE,50,[0,15,30,0,0,0,0,0,0],[0,0,0,0,0,0,0]];

    !TouchMotion
    PERS bool bTouchError{4,2}:=[[FALSE,FALSE],[FALSE,FALSE],[FALSE,FALSE],[FALSE,FALSE]];
    PERS num nCheckCount:=1;
    PERS num RetryDepthData{3}:=[10,-10,10];
    PERS bool bRetry:=FALSE;
    PERS string TouchErrorDirMain:="Ready";
    PERS string TouchErrorDirSub:="Ready";
    PERS jointgroup jSearchReadyGroup;
    PERS pointgroup pSearchReadyGroup;
    PERS jointtarget jSearchReady:=[[9E+09,9E+09,9E+09,9E+09,9E+09,9E+09],[10404,5130.4,470.866,89.8328,9E+09,10404]];
    PERS num nArcErrorPos:=0;
    PERS robtarget pArcErrorPos:=[[6,8,12],[1,0,0,0],[0,0,0,0],[0,0,0,0,9E+09,9E+09]];
    PERS bool bTouchWorkCount{6};
    PERS bool bEndSearchComplete:=FALSE;
    PERS bool bSumTouchError:=FALSE;

    !Arc_Error
    PERS bool bArcError:=FALSE;

    !! Variables for HoleSensor based Origin Checking
    PERS num nRefHoleX{2}:=[5.7,0.4];
    PERS num nInspectHoleX{2}:=[6.05,0.33];
    PERS num nDiffHoleX:=0.35;
    PERS num nDiffHoleXskew:=-0.00273613;

    !! Variables for LDS based Origin Checking
    CONST pos pInspectGantryOriginal:=[2054.978,731.4054,1208.162];
    PERS num nInspectGantryX{2}:=[7178.18,7178.38];
    PERS num nInspectGantryY{2}:=[569.71,569.63];
    PERS num nInspectGantryZ{2}:=[475.415,475.436];
    PERS num nDiffGantryX:=0;
    PERS num nDiffGantryY:=0;
    PERS num nDiffGantryZ:=0;

    PERS num nCorrX_Store_Start{2};
    PERS num nCorrY_Store_Start{2};
    PERS num nCorrZ_Store_Start{2};
    PERS num nCorrX_Store_End{2};
    PERS num nCorrY_Store_End{2};
    PERS num nCorrZ_Store_End{2};

    PERS seamdata smDefault_1{2};
    PERS seamdata seam_TRob1;
    PERS seamdata smDefault_2{2};
    PERS seamdata seam_TRob2;

    ! Variables for Touch Sync
    PERS bool bTouch_last_R1_Comp:=TRUE;
    PERS bool bTouch_last_R2_Comp:=TRUE;
    PERS bool bTouch_First_R1_Comp:=TRUE;
    PERS bool bTouch_First_R2_Comp:=TRUE;
    PERS bool bGanTry_First_pos:=FALSE;
    PERS bool bGanTry_Last_pos:=FALSE;

    PERS jointtarget jCorrT_ROB1_Start;
    PERS jointtarget jCorrT_ROB1_End;
    PERS robtarget pCorrT_ROB1_Start;
    PERS robtarget pCorrT_ROB1_End;

    PERS robtarget pCorrT_ROB2_Start;
    PERS robtarget pCorrT_ROB2_End;
    PERS jointtarget jCorrTouchGantry_Start;
    PERS jointtarget jCorrTouchGantry_End;
    PERS tooldata tWeld1copy:=[TRUE,[[320.377,0,330.247],[0.92587,0,0.37784,0]],[3.1,[-71.4,3.8,173.2],[1,0,0,0],0.055,0.049,0.005]];
    PERS tooldata tWeldcopy2:=[TRUE,[[308.188,-16.1693,300.214],[0.92587,0,0.37784,0]],[3.1,[-71.4,3.8,173.2],[1,0,0,0],0.055,0.049,0.005]];
    PERS targetdata Welds1{40}:=[[[[0,9.09738,4.25871],[0.241845,0.664463,-0.664463,0.241845],[0,0,0,1],[9E+09,9E+09,9E+09,9E+09,9E+09,9E+09]],60,0,36.8,230,380,1,2,2,1.5,1,1,0,0,0,0,0],[[[1,9.09738,4.25871],[0.241845,0.664463,-0.664463,0.241845],[0,0,0,1],[9E+09,9E+09,9E+09,9E+09,9E+09,9E+09]],60,0,36.8,230,380,1,2,2,1.5,1,1,0,0,0,0,0],[[[2,9.09738,4.25871],[0.241845,0.664463,-0.664463,0.241845],[0,0,0,1],[9E+09,9E+09,9E+09,9E+09,9E+09,9E+09]],60,0,36.8,230,380,1,2,2,1.5,1,1,0,0,0,0,0],[[[3,9.09738,4.25871],[0.241845,0.664463,-0.664463,0.241845],[0,0,0,1],[9E+09,9E+09,9E+09,9E+09,9E+09,9E+09]],60,0,36.8,230,380,1,2,2,1.5,1,1,0,0,0,0,0],[[[25,9.09738,4.25871],[0.241845,0.664463,-0.664463,0.241845],[0,0,0,1],[9E+09,9E+09,9E+09,9E+09,9E+09,9E+09]],60,0,36.8,230,380,1,2,2,1.5,1,1,0,10,20,0,0],[[[75,4.68064,1.11234],[0.241845,0.664463,-0.664463,0.241845],[0,0,0,1],[9E+09,9E+09,9E+09,9E+09,9E+09,9E+09]],60,0,36.8,230,380,1,2,2,1.5,1,1,0,10,20,0,0],[[[97,4.68064,1.11234],[0.241845,0.664463,-0.664463,0.241845],[0,0,0,1],[9E+09,9E+09,9E+09,9E+09,9E+09,9E+09]],60,0,36.8,230,380,1,2,2,1.5,1,1,0,10,20,0,0],[[[98,4.68064,1.11234],[0.241845,0.664463,-0.664463,0.241845],[0,0,0,1],[9E+09,9E+09,9E+09,9E+09,9E+09,9E+09]],60,0,36.8,230,380,1,2,2,1.5,1,1,0,0,0,0,0],[[[99,4.68064,1.11234],[0.241845,0.664463,-0.664463,0.241845],[0,0,0,1],[9E+09,9E+09,9E+09,9E+09,9E+09,9E+09]],60,0,36.8,230,380,1,2,2,1.5,1,1,0,0,0,0,0],[[[100,4.68064,1.11234],[0.241845,0.664463,-0.664463,0.241845],[0,0,0,1],[9E+09,9E+09,9E+09,9E+09,9E+09,9E+09]],60,0,36.8,230,380,1,2,2,1.5,1,1,0,0,0,0,0],[[[0,0,0],[1,0,0,0],[0,0,0,0],[9E+09,9E+09,9E+09,9E+09,9E+09,9E+09]],0,0,0,0,0,0,0,0,0,0,0,0,0,0,0,0],[[[0,0,0],[1,0,0,0],[0,0,0,0],[9E+09,9E+09,9E+09,9E+09,9E+09,9E+09]],0,0,0,0,0,0,0,0,0,0,0,0,0,0,0,0],[[[0,0,0],[1,0,0,0],[0,0,0,0],[9E+09,9E+09,9E+09,9E+09,9E+09,9E+09]],0,0,0,0,0,0,0,0,0,0,0,0,0,0,0,0],[[[0,0,0],[1,0,0,0],[0,0,0,0],[9E+09,9E+09,9E+09,9E+09,9E+09,9E+09]],0,0,0,0,0,0,0,0,0,0,0,0,0,0,0,0],[[[0,0,0],[1,0,0,0],[0,0,0,0],[9E+09,9E+09,9E+09,9E+09,9E+09,9E+09]],0,0,0,0,0,0,0,0,0,0,0,0,0,0,0,0],[[[0,0,0],[1,0,0,0],[0,0,0,0],[9E+09,9E+09,9E+09,9E+09,9E+09,9E+09]],0,0,0,0,0,0,0,0,0,0,0,0,0,0,0,0],[[[0,0,0],[1,0,0,0],[0,0,0,0],[9E+09,9E+09,9E+09,9E+09,9E+09,9E+09]],0,0,0,0,0,0,0,0,0,0,0,0,0,0,0,0],[[[0,0,0],[1,0,0,0],[0,0,0,0],[9E+09,9E+09,9E+09,9E+09,9E+09,9E+09]],0,0,0,0,0,0,0,0,0,0,0,0,0,0,0,0],[[[0,0,0],[1,0,0,0],[0,0,0,0],[9E+09,9E+09,9E+09,9E+09,9E+09,9E+09]],0,0,0,0,0,0,0,0,0,0,0,0,0,0,0,0],[[[0,0,0],[1,0,0,0],[0,0,0,0],[9E+09,9E+09,9E+09,9E+09,9E+09,9E+09]],0,0,0,0,0,0,0,0,0,0,0,0,0,0,0,0],[[[0,0,0],[1,0,0,0],[0,0,0,0],[9E+09,9E+09,9E+09,9E+09,9E+09,9E+09]],0,0,0,0,0,0,0,0,0,0,0,0,0,0,0,0],[[[0,0,0],[1,0,0,0],[0,0,0,0],[9E+09,9E+09,9E+09,9E+09,9E+09,9E+09]],0,0,0,0,0,0,0,0,0,0,0,0,0,0,0,0],[[[0,0,0],[1,0,0,0],[0,0,0,0],[9E+09,9E+09,9E+09,9E+09,9E+09,9E+09]],0,0,0,0,0,0,0,0,0,0,0,0,0,0,0,0],[[[0,0,0],[1,0,0,0],[0,0,0,0],[9E+09,9E+09,9E+09,9E+09,9E+09,9E+09]],0,0,0,0,0,0,0,0,0,0,0,0,0,0,0,0],[[[0,0,0],[1,0,0,0],[0,0,0,0],[9E+09,9E+09,9E+09,9E+09,9E+09,9E+09]],0,0,0,0,0,0,0,0,0,0,0,0,0,0,0,0],[[[0,0,0],[1,0,0,0],[0,0,0,0],[9E+09,9E+09,9E+09,9E+09,9E+09,9E+09]],0,0,0,0,0,0,0,0,0,0,0,0,0,0,0,0],[[[0,0,0],[1,0,0,0],[0,0,0,0],[9E+09,9E+09,9E+09,9E+09,9E+09,9E+09]],0,0,0,0,0,0,0,0,0,0,0,0,0,0,0,0],[[[0,0,0],[1,0,0,0],[0,0,0,0],[9E+09,9E+09,9E+09,9E+09,9E+09,9E+09]],0,0,0,0,0,0,0,0,0,0,0,0,0,0,0,0],[[[0,0,0],[1,0,0,0],[0,0,0,0],[9E+09,9E+09,9E+09,9E+09,9E+09,9E+09]],0,0,0,0,0,0,0,0,0,0,0,0,0,0,0,0],[[[0,0,0],[1,0,0,0],[0,0,0,0],[9E+09,9E+09,9E+09,9E+09,9E+09,9E+09]],0,0,0,0,0,0,0,0,0,0,0,0,0,0,0,0],[[[0,0,0],[1,0,0,0],[0,0,0,0],[9E+09,9E+09,9E+09,9E+09,9E+09,9E+09]],0,0,0,0,0,0,0,0,0,0,0,0,0,0,0,0],[[[0,0,0],[1,0,0,0],[0,0,0,0],[9E+09,9E+09,9E+09,9E+09,9E+09,9E+09]],0,0,0,0,0,0,0,0,0,0,0,0,0,0,0,0],[[[0,0,0],[1,0,0,0],[0,0,0,0],[9E+09,9E+09,9E+09,9E+09,9E+09,9E+09]],0,0,0,0,0,0,0,0,0,0,0,0,0,0,0,0],[[[0,0,0],[1,0,0,0],[0,0,0,0],[9E+09,9E+09,9E+09,9E+09,9E+09,9E+09]],0,0,0,0,0,0,0,0,0,0,0,0,0,0,0,0],[[[0,0,0],[1,0,0,0],[0,0,0,0],[9E+09,9E+09,9E+09,9E+09,9E+09,9E+09]],0,0,0,0,0,0,0,0,0,0,0,0,0,0,0,0],[[[0,0,0],[1,0,0,0],[0,0,0,0],[9E+09,9E+09,9E+09,9E+09,9E+09,9E+09]],0,0,0,0,0,0,0,0,0,0,0,0,0,0,0,0],[[[0,0,0],[1,0,0,0],[0,0,0,0],[9E+09,9E+09,9E+09,9E+09,9E+09,9E+09]],0,0,0,0,0,0,0,0,0,0,0,0,0,0,0,0],[[[0,0,0],[1,0,0,0],[0,0,0,0],[9E+09,9E+09,9E+09,9E+09,9E+09,9E+09]],0,0,0,0,0,0,0,0,0,0,0,0,0,0,0,0],[[[0,0,0],[1,0,0,0],[0,0,0,0],[9E+09,9E+09,9E+09,9E+09,9E+09,9E+09]],0,0,0,0,0,0,0,0,0,0,0,0,0,0,0,0],[[[0,0,0],[1,0,0,0],[0,0,0,0],[9E+09,9E+09,9E+09,9E+09,9E+09,9E+09]],0,0,0,0,0,0,0,0,0,0,0,0,0,0,0,0]];
    PERS targetdata Welds2{40}:=[[[[0,-9.76043,2.19295],[0.241845,-0.664463,-0.664463,-0.241845],[0,0,0,1],[9E+09,9E+09,9E+09,9E+09,9E+09,9E+09]],60,0,36.3,232,360,1,2,2,1.5,1,1,0,0,0,0,0],[[[1,-9.76043,2.19295],[0.241845,-0.664463,-0.664463,-0.241845],[0,0,0,1],[9E+09,9E+09,9E+09,9E+09,9E+09,9E+09]],60,0,36.3,232,360,1,2,2,1.5,1,1,0,0,0,0,0],[[[2,-9.76043,2.19295],[0.241845,-0.664463,-0.664463,-0.241845],[0,0,0,1],[9E+09,9E+09,9E+09,9E+09,9E+09,9E+09]],60,0,36.3,232,360,1,2,2,1.5,1,1,0,0,0,0,0],[[[3,-9.76043,2.19295],[0.241845,-0.664463,-0.664463,-0.241845],[0,0,0,1],[9E+09,9E+09,9E+09,9E+09,9E+09,9E+09]],60,0,36.3,232,360,1,2,2,1.5,1,1,0,0,0,0,0],[[[25,-9.76043,2.19295],[0.241845,-0.664463,-0.664463,-0.241845],[0,0,0,1],[9E+09,9E+09,9E+09,9E+09,9E+09,9E+09]],60,0,36.3,232,360,1,2,2,1.5,1,1,0,10,20,0,0],[[[75,-13.4213,-1.06604],[0.241845,-0.664463,-0.664463,-0.241845],[0,0,0,1],[9E+09,9E+09,9E+09,9E+09,9E+09,9E+09]],60,0,36.3,232,360,1,2,2,1.5,1,1,0,10,20,0,0],[[[97,-13.4213,-1.06604],[0.241845,-0.664463,-0.664463,-0.241845],[0,0,0,1],[9E+09,9E+09,9E+09,9E+09,9E+09,9E+09]],60,0,36.3,232,360,1,2,2,1.5,1,1,0,10,20,0,0],[[[98,-13.4213,-1.06604],[0.241845,-0.664463,-0.664463,-0.241845],[0,0,0,1],[9E+09,9E+09,9E+09,9E+09,9E+09,9E+09]],60,0,36.3,232,360,1,2,2,1.5,1,1,0,0,0,0,0],[[[99,-12.4213,-1.06604],[0.241845,-0.664463,-0.664463,-0.241845],[0,0,0,1],[9E+09,9E+09,9E+09,9E+09,9E+09,9E+09]],60,0,36.3,232,360,1,2,2,1.5,1,1,0,0,0,0,0],[[[100,-12.4213,-1.06604],[0.241845,-0.664463,-0.664463,-0.241845],[0,0,0,1],[9E+09,9E+09,9E+09,9E+09,9E+09,9E+09]],60,0,36.3,232,360,1,2,2,1.5,1,1,0,0,0,0,0],[[[0,0,0],[1,0,0,0],[0,0,0,0],[9E+09,9E+09,9E+09,9E+09,9E+09,9E+09]],0,0,0,0,0,0,0,0,0,0,0,0,0,0,0,0],[[[0,0,0],[1,0,0,0],[0,0,0,0],[9E+09,9E+09,9E+09,9E+09,9E+09,9E+09]],0,0,0,0,0,0,0,0,0,0,0,0,0,0,0,0],[[[0,0,0],[1,0,0,0],[0,0,0,0],[9E+09,9E+09,9E+09,9E+09,9E+09,9E+09]],0,0,0,0,0,0,0,0,0,0,0,0,0,0,0,0],[[[0,0,0],[1,0,0,0],[0,0,0,0],[9E+09,9E+09,9E+09,9E+09,9E+09,9E+09]],0,0,0,0,0,0,0,0,0,0,0,0,0,0,0,0],[[[0,0,0],[1,0,0,0],[0,0,0,0],[9E+09,9E+09,9E+09,9E+09,9E+09,9E+09]],0,0,0,0,0,0,0,0,0,0,0,0,0,0,0,0],[[[0,0,0],[1,0,0,0],[0,0,0,0],[9E+09,9E+09,9E+09,9E+09,9E+09,9E+09]],0,0,0,0,0,0,0,0,0,0,0,0,0,0,0,0],[[[0,0,0],[1,0,0,0],[0,0,0,0],[9E+09,9E+09,9E+09,9E+09,9E+09,9E+09]],0,0,0,0,0,0,0,0,0,0,0,0,0,0,0,0],[[[0,0,0],[1,0,0,0],[0,0,0,0],[9E+09,9E+09,9E+09,9E+09,9E+09,9E+09]],0,0,0,0,0,0,0,0,0,0,0,0,0,0,0,0],[[[0,0,0],[1,0,0,0],[0,0,0,0],[9E+09,9E+09,9E+09,9E+09,9E+09,9E+09]],0,0,0,0,0,0,0,0,0,0,0,0,0,0,0,0],[[[0,0,0],[1,0,0,0],[0,0,0,0],[9E+09,9E+09,9E+09,9E+09,9E+09,9E+09]],0,0,0,0,0,0,0,0,0,0,0,0,0,0,0,0],[[[0,0,0],[1,0,0,0],[0,0,0,0],[9E+09,9E+09,9E+09,9E+09,9E+09,9E+09]],0,0,0,0,0,0,0,0,0,0,0,0,0,0,0,0],[[[0,0,0],[1,0,0,0],[0,0,0,0],[9E+09,9E+09,9E+09,9E+09,9E+09,9E+09]],0,0,0,0,0,0,0,0,0,0,0,0,0,0,0,0],[[[0,0,0],[1,0,0,0],[0,0,0,0],[9E+09,9E+09,9E+09,9E+09,9E+09,9E+09]],0,0,0,0,0,0,0,0,0,0,0,0,0,0,0,0],[[[0,0,0],[1,0,0,0],[0,0,0,0],[9E+09,9E+09,9E+09,9E+09,9E+09,9E+09]],0,0,0,0,0,0,0,0,0,0,0,0,0,0,0,0],[[[0,0,0],[1,0,0,0],[0,0,0,0],[9E+09,9E+09,9E+09,9E+09,9E+09,9E+09]],0,0,0,0,0,0,0,0,0,0,0,0,0,0,0,0],[[[0,0,0],[1,0,0,0],[0,0,0,0],[9E+09,9E+09,9E+09,9E+09,9E+09,9E+09]],0,0,0,0,0,0,0,0,0,0,0,0,0,0,0,0],[[[0,0,0],[1,0,0,0],[0,0,0,0],[9E+09,9E+09,9E+09,9E+09,9E+09,9E+09]],0,0,0,0,0,0,0,0,0,0,0,0,0,0,0,0],[[[0,0,0],[1,0,0,0],[0,0,0,0],[9E+09,9E+09,9E+09,9E+09,9E+09,9E+09]],0,0,0,0,0,0,0,0,0,0,0,0,0,0,0,0],[[[0,0,0],[1,0,0,0],[0,0,0,0],[9E+09,9E+09,9E+09,9E+09,9E+09,9E+09]],0,0,0,0,0,0,0,0,0,0,0,0,0,0,0,0],[[[0,0,0],[1,0,0,0],[0,0,0,0],[9E+09,9E+09,9E+09,9E+09,9E+09,9E+09]],0,0,0,0,0,0,0,0,0,0,0,0,0,0,0,0],[[[0,0,0],[1,0,0,0],[0,0,0,0],[9E+09,9E+09,9E+09,9E+09,9E+09,9E+09]],0,0,0,0,0,0,0,0,0,0,0,0,0,0,0,0],[[[0,0,0],[1,0,0,0],[0,0,0,0],[9E+09,9E+09,9E+09,9E+09,9E+09,9E+09]],0,0,0,0,0,0,0,0,0,0,0,0,0,0,0,0],[[[0,0,0],[1,0,0,0],[0,0,0,0],[9E+09,9E+09,9E+09,9E+09,9E+09,9E+09]],0,0,0,0,0,0,0,0,0,0,0,0,0,0,0,0],[[[0,0,0],[1,0,0,0],[0,0,0,0],[9E+09,9E+09,9E+09,9E+09,9E+09,9E+09]],0,0,0,0,0,0,0,0,0,0,0,0,0,0,0,0],[[[0,0,0],[1,0,0,0],[0,0,0,0],[9E+09,9E+09,9E+09,9E+09,9E+09,9E+09]],0,0,0,0,0,0,0,0,0,0,0,0,0,0,0,0],[[[0,0,0],[1,0,0,0],[0,0,0,0],[9E+09,9E+09,9E+09,9E+09,9E+09,9E+09]],0,0,0,0,0,0,0,0,0,0,0,0,0,0,0,0],[[[0,0,0],[1,0,0,0],[0,0,0,0],[9E+09,9E+09,9E+09,9E+09,9E+09,9E+09]],0,0,0,0,0,0,0,0,0,0,0,0,0,0,0,0],[[[0,0,0],[1,0,0,0],[0,0,0,0],[9E+09,9E+09,9E+09,9E+09,9E+09,9E+09]],0,0,0,0,0,0,0,0,0,0,0,0,0,0,0,0],[[[0,0,0],[1,0,0,0],[0,0,0,0],[9E+09,9E+09,9E+09,9E+09,9E+09,9E+09]],0,0,0,0,0,0,0,0,0,0,0,0,0,0,0,0],[[[0,0,0],[1,0,0,0],[0,0,0,0],[9E+09,9E+09,9E+09,9E+09,9E+09,9E+09]],0,0,0,0,0,0,0,0,0,0,0,0,0,0,0,0]];
    PERS targetdata WeldsG{40}:=[[[[19996.4,2731.64,1624.12],[0.708156,0,0,-0.706056],[0,0,0,0],[9E+09,9E+09,9E+09,9E+09,9E+09,9E+09]],0,0,0,0,0,0,0,0,0,0,0,0,0,0,0,0],[[[20004,169.605,1622.71],[0.708156,0,0,-0.706056],[0,0,0,0],[9E+09,9E+09,9E+09,9E+09,9E+09,9E+09]],0,0,0,0,0,0,0,0,0,0,0,0,0,0,0,0],[[[0,0,0],[1,0,0,0],[0,0,0,0],[9E+09,9E+09,9E+09,9E+09,9E+09,9E+09]],0,0,0,0,0,0,0,0,0,0,0,0,0,0,0,0],[[[0,0,0],[1,0,0,0],[0,0,0,0],[9E+09,9E+09,9E+09,9E+09,9E+09,9E+09]],0,0,0,0,0,0,0,0,0,0,0,0,0,0,0,0],[[[0,0,0],[1,0,0,0],[0,0,0,0],[9E+09,9E+09,9E+09,9E+09,9E+09,9E+09]],0,0,0,0,0,0,0,0,0,0,0,0,0,0,0,0],[[[0,0,0],[1,0,0,0],[0,0,0,0],[9E+09,9E+09,9E+09,9E+09,9E+09,9E+09]],0,0,0,0,0,0,0,0,0,0,0,0,0,0,0,0],[[[0,0,0],[1,0,0,0],[0,0,0,0],[9E+09,9E+09,9E+09,9E+09,9E+09,9E+09]],0,0,0,0,0,0,0,0,0,0,0,0,0,0,0,0],[[[0,0,0],[1,0,0,0],[0,0,0,0],[9E+09,9E+09,9E+09,9E+09,9E+09,9E+09]],0,0,0,0,0,0,0,0,0,0,0,0,0,0,0,0],[[[0,0,0],[1,0,0,0],[0,0,0,0],[9E+09,9E+09,9E+09,9E+09,9E+09,9E+09]],0,0,0,0,0,0,0,0,0,0,0,0,0,0,0,0],[[[0,0,0],[1,0,0,0],[0,0,0,0],[9E+09,9E+09,9E+09,9E+09,9E+09,9E+09]],0,0,0,0,0,0,0,0,0,0,0,0,0,0,0,0],[[[0,0,0],[1,0,0,0],[0,0,0,0],[9E+09,9E+09,9E+09,9E+09,9E+09,9E+09]],0,0,0,0,0,0,0,0,0,0,0,0,0,0,0,0],[[[0,0,0],[1,0,0,0],[0,0,0,0],[9E+09,9E+09,9E+09,9E+09,9E+09,9E+09]],0,0,0,0,0,0,0,0,0,0,0,0,0,0,0,0],[[[0,0,0],[1,0,0,0],[0,0,0,0],[9E+09,9E+09,9E+09,9E+09,9E+09,9E+09]],0,0,0,0,0,0,0,0,0,0,0,0,0,0,0,0],[[[0,0,0],[1,0,0,0],[0,0,0,0],[9E+09,9E+09,9E+09,9E+09,9E+09,9E+09]],0,0,0,0,0,0,0,0,0,0,0,0,0,0,0,0],[[[0,0,0],[1,0,0,0],[0,0,0,0],[9E+09,9E+09,9E+09,9E+09,9E+09,9E+09]],0,0,0,0,0,0,0,0,0,0,0,0,0,0,0,0],[[[0,0,0],[1,0,0,0],[0,0,0,0],[9E+09,9E+09,9E+09,9E+09,9E+09,9E+09]],0,0,0,0,0,0,0,0,0,0,0,0,0,0,0,0],[[[0,0,0],[1,0,0,0],[0,0,0,0],[9E+09,9E+09,9E+09,9E+09,9E+09,9E+09]],0,0,0,0,0,0,0,0,0,0,0,0,0,0,0,0],[[[0,0,0],[1,0,0,0],[0,0,0,0],[9E+09,9E+09,9E+09,9E+09,9E+09,9E+09]],0,0,0,0,0,0,0,0,0,0,0,0,0,0,0,0],[[[0,0,0],[1,0,0,0],[0,0,0,0],[9E+09,9E+09,9E+09,9E+09,9E+09,9E+09]],0,0,0,0,0,0,0,0,0,0,0,0,0,0,0,0],[[[0,0,0],[1,0,0,0],[0,0,0,0],[9E+09,9E+09,9E+09,9E+09,9E+09,9E+09]],0,0,0,0,0,0,0,0,0,0,0,0,0,0,0,0],[[[0,0,0],[1,0,0,0],[0,0,0,0],[9E+09,9E+09,9E+09,9E+09,9E+09,9E+09]],0,0,0,0,0,0,0,0,0,0,0,0,0,0,0,0],[[[0,0,0],[1,0,0,0],[0,0,0,0],[9E+09,9E+09,9E+09,9E+09,9E+09,9E+09]],0,0,0,0,0,0,0,0,0,0,0,0,0,0,0,0],[[[0,0,0],[1,0,0,0],[0,0,0,0],[9E+09,9E+09,9E+09,9E+09,9E+09,9E+09]],0,0,0,0,0,0,0,0,0,0,0,0,0,0,0,0],[[[0,0,0],[1,0,0,0],[0,0,0,0],[9E+09,9E+09,9E+09,9E+09,9E+09,9E+09]],0,0,0,0,0,0,0,0,0,0,0,0,0,0,0,0],[[[0,0,0],[1,0,0,0],[0,0,0,0],[9E+09,9E+09,9E+09,9E+09,9E+09,9E+09]],0,0,0,0,0,0,0,0,0,0,0,0,0,0,0,0],[[[0,0,0],[1,0,0,0],[0,0,0,0],[9E+09,9E+09,9E+09,9E+09,9E+09,9E+09]],0,0,0,0,0,0,0,0,0,0,0,0,0,0,0,0],[[[0,0,0],[1,0,0,0],[0,0,0,0],[9E+09,9E+09,9E+09,9E+09,9E+09,9E+09]],0,0,0,0,0,0,0,0,0,0,0,0,0,0,0,0],[[[0,0,0],[1,0,0,0],[0,0,0,0],[9E+09,9E+09,9E+09,9E+09,9E+09,9E+09]],0,0,0,0,0,0,0,0,0,0,0,0,0,0,0,0],[[[0,0,0],[1,0,0,0],[0,0,0,0],[9E+09,9E+09,9E+09,9E+09,9E+09,9E+09]],0,0,0,0,0,0,0,0,0,0,0,0,0,0,0,0],[[[0,0,0],[1,0,0,0],[0,0,0,0],[9E+09,9E+09,9E+09,9E+09,9E+09,9E+09]],0,0,0,0,0,0,0,0,0,0,0,0,0,0,0,0],[[[0,0,0],[1,0,0,0],[0,0,0,0],[9E+09,9E+09,9E+09,9E+09,9E+09,9E+09]],0,0,0,0,0,0,0,0,0,0,0,0,0,0,0,0],[[[0,0,0],[1,0,0,0],[0,0,0,0],[9E+09,9E+09,9E+09,9E+09,9E+09,9E+09]],0,0,0,0,0,0,0,0,0,0,0,0,0,0,0,0],[[[0,0,0],[1,0,0,0],[0,0,0,0],[9E+09,9E+09,9E+09,9E+09,9E+09,9E+09]],0,0,0,0,0,0,0,0,0,0,0,0,0,0,0,0],[[[0,0,0],[1,0,0,0],[0,0,0,0],[9E+09,9E+09,9E+09,9E+09,9E+09,9E+09]],0,0,0,0,0,0,0,0,0,0,0,0,0,0,0,0],[[[0,0,0],[1,0,0,0],[0,0,0,0],[9E+09,9E+09,9E+09,9E+09,9E+09,9E+09]],0,0,0,0,0,0,0,0,0,0,0,0,0,0,0,0],[[[0,0,0],[1,0,0,0],[0,0,0,0],[9E+09,9E+09,9E+09,9E+09,9E+09,9E+09]],0,0,0,0,0,0,0,0,0,0,0,0,0,0,0,0],[[[0,0,0],[1,0,0,0],[0,0,0,0],[9E+09,9E+09,9E+09,9E+09,9E+09,9E+09]],0,0,0,0,0,0,0,0,0,0,0,0,0,0,0,0],[[[0,0,0],[1,0,0,0],[0,0,0,0],[9E+09,9E+09,9E+09,9E+09,9E+09,9E+09]],0,0,0,0,0,0,0,0,0,0,0,0,0,0,0,0],[[[0,0,0],[1,0,0,0],[0,0,0,0],[9E+09,9E+09,9E+09,9E+09,9E+09,9E+09]],0,0,0,0,0,0,0,0,0,0,0,0,0,0,0,0],[[[0,0,0],[1,0,0,0],[0,0,0,0],[9E+09,9E+09,9E+09,9E+09,9E+09,9E+09]],0,0,0,0,0,0,0,0,0,0,0,0,0,0,0,0]];
    PERS bool bMoveHome_Head;
    !Error
    PERS num nErrorCmd;
    !Error_Pos
    PERS num nWeldDist;
    PERS monRobs MonitorweldErrorpostion;
    PERS num nEntryRetryCount{2}:=[0,0];
    PERS num nTouchRetryCount{2}:=[0,0];
    PERS bool bGantryInTrap{2};
    PERS num nWeldLineLength_R1;
    PERS num nWeldLineLength_R2;
    PERS num nMaintenanceYPos:=5300;
    PERS num nInchingTime:=2.1;
    PERS bool bGUI_ArcRefresh;
    PERS bool bBreakPoint{2};
    PERS num nBreakPoint{2};
    PERS bool btouchTimeOut{2}:=[FALSE,FALSE];
    PERS bool bWeldOutputDisable:=TRUE;
    PERS bool bso_MoveG_PosHold:=FALSE;
    PERS num nMoveid:=1;
    PERS bool bRBT_PP_Main:=FALSE;
    PERS bool bWireCutSync:=FALSE;
    !!!!!!!!!
    PERS jointgroup jgMeasurementHome:=[[[40,90,-90,0,0,0],[9E+09,9E+09,9E+09,9E+09,9E+09,9E+09]],[[40,90,-90,0,0,0],[9E+09,9E+09,9E+09,9E+09,9E+09,9E+09]],[[9E+09,9E+09,9E+09,9E+09,9E+09,9E+09],[7000,5300,0,0,9E+09,7000]]];
    PERS jointgroup jgWireCutHome:=[[[39.7077,23.0399,30.4536,-87.5281,29.1211,122.951],[9E+09,9E+09,9E+09,9E+09,9E+09,9E+09]],[[39.5269,22.7659,30.4413,-87.1375,29.0323,122.34],[9E+09,9E+09,9E+09,9E+09,9E+09,9E+09]],[[9E+09,9E+09,9E+09,9E+09,9E+09,9E+09],[7000,5300,0,0,9E+09,7000]]];
    PERS bool bWirecut{3}:=[FALSE,TRUE,FALSE];
    PERS bool bArc_On{2}:=[FALSE,FALSE];

    PERS num nOffsetStart_Gantry:=50;
    PERS num nOffsetEnd_Gantry:=50;

    PERS num nOffsetStart_A:=50;
    PERS num nOffsetEnd_A:=50;
    PERS num nOffsetStart_B:=50;
    PERS num nOffsetEnd_B:=50;

    PERS num nOffsetStartBuffer:=0;
    PERS num nOffsetEndBuffer:=0;
    PERS num nMode:=3;
    PERS num nWarmUpCycle:=600;
    PERS jointgroup jgWarm_Up;
    PERS jointgroup jgTarget;
    PERS num nWarmUpTime:=599.626;

    !======== Tcp Check
    PERS TcpOrder tOrder:=[4000,3300,150,90];
    PERS jointgroup jgMoveToTcp;
    PERS jointgroup jgMoveToTcpComparison;
    !!! Retry
    pers num nTouchWhileMovingCount_R1;
    pers num nTouchWhileMovingCount_R2;
    pers bool bTouchOnSameSpotError_R1;
    pers bool bTouchOnSameSpotError_R2;
    PERS num nSameSpot_StartX_R1:=0;
    PERS num nSameSpot_StartY_R1:=0;
    PERS num nSameSpot_StartZ_R1:=0;
    PERS num nSameSpot_EndX_R1:=0;
    PERS num nSameSpot_EndY_R1:=0;
    PERS num nSameSpot_EndZ_R1:=0;
    PERS num nSameSpot_StartX_R2:=0;
    PERS num nSameSpot_StartY_R2:=0;
    PERS num nSameSpot_StartZ_R2:=0;
    PERS num nSameSpot_EndX_R2:=0;
    PERS num nSameSpot_EndY_R2:=0;
    PERS num nSameSpot_EndZ_R2:=0;
    PERS bool bMoveToWireCutHome:=TRUE;

    PERS num nSprayTime:=1;
    PERS jointtarget jNozzleClean_R1;
    PERS jointtarget jNozzleClean_R2;
    PERS bool bNozzleCleanCut:=FALSE;
    PERS num nR_Angle:=90;

    PERS num nSearchBuffer_X_Start{2};
    PERS num nSearchBuffer_Y_Start{2};
    PERS num nSearchBuffer_Z_Start{2};
    PERS num nSearchBuffer_X_End{2};
    PERS num nSearchBuffer_Y_End{2};
    PERS num nSearchBuffer_Z_End{2};
    !!!!!  TeachingWireCut  !!!!!!!!!!!!!
    PERS pos pCuttingInsideOffset_R1;
    PERS pos pCuttingInsideOffset_R2;
    PERS pos pCuttingEntryOffset_R1;
    PERS pos pCuttingEntryOffset_R2;
    PERS bool bTeachingWireCut:=FALSE;

    !!! Variables for Hole/LDS Inspect
    PERS bool bHoleCheckScss;
    PERS bool bLDSCheckScss;

ENDMODULE
